(* CODESYS project oakslibrary.library
   Title: OaksLibrary
   Version: 1.1
   Placeholder: OaksLibrary
   Company: OaksAB

Project tree, tasks and I/O mapping:
  libraries: Tc2_BA, 3.3.9.0 (Beckhoff Automation GmbH); Tc2_EtherCAT, * (Beckhoff Automation GmbH); Tc2_IoFunctions, 3.3.13.0 (Beckhoff Automation GmbH); Tc2_Standard, 3.3.3.0 (Beckhoff Automation GmbH); Tc2_SUPS, 3.3.8.0 (Beckhoff Automation GmbH); Tc2_System, 3.4.24.0 (Beckhoff Automation GmbH); Tc2_SystemCX, 3.3.6.0 (Beckhoff Automation GmbH); Tc2_Utilities, * (Beckhoff Automation GmbH); Tc3_BA, 1.1.5.0 (Beckhoff Automation GmbH); Tc3_BA_Common, 2.1.4.0 (Beckhoff Automation GmbH); Tc3_Module, 3.3.21.0 (Beckhoff Automation GmbH)
  oaksLibrary/
    1 Ej vidareutveckling/
      function block fbDewpoint [ST]
      function block fbModbusSekvens [ST]
      function fRealToHour [CFC]
      function fRealToMinute [CFC]
      function fRealToSecond [CFC]
    Beräkning/
      Närvaro/
        function block fbCalcPresenceCo2Flow [ST]
        function fCalcPresenceCo2Flow [ST]
      function fAverageValueCalc [ST]
      function block fbCopCalc [ST]
      function block fbDewpointCalc [ST]
      function block fbDewPointSafe [ST]
      function block fbDifferenceCheck [ST]
      function block fbHeatExhEfficiency [ST]
      function block fbHourDiff [ST]
      function block fbMeanValueBC [ST]
      function block fbOperatingHours [ST]
      function block fbScale6pSupTempRad [ST]
      function block fbScale6pSuptempVent [ST]
      function block fbSfpCalc [ST]
      function block fbSunClock [ST]: DAY_OF_YEAR, DEG, FLOOR2, HOUR, HOUR_TO_TIME, HOUR_TO_TOD, MINUTE, MODR, mPercentageOfDay, mSolnedOchUppGangForskjuten, mSoluppgangOchSolnedgang, RAD, SUN_MIDDAY
      function fCalcFlow [ST]
      function fCalcFlowfbNicotraGerbhardtRLM [ST]
      function fScale12pInternalSetpoint [ST]
      function fScale20p [ST]
      function fScale2p [ST]
      function fScale2pInternalSetpoint [ST]
      function fScale3p [ST]
      function fScale3pInternalSetpoint [ST]
      function fScale6p [ST]
      function fScale6pInternalSetpoint [ST]
      function fScale7p [ST]
      function fScale7pInternalSetpoint [ST]
    Brand/
      function block fbFirealarm [ST]
      function block fbFirealarmFailure [ST]
      function block fbFireDamper [ST]
      function block fbFireDamperEvac [ST]
      function block fbFiredamperExercise [ST]
      function block fbFireDamperOneInput [ST]
      function block fbFireDamperWithAnalogOutput [ST]
      function block fbSmokeDetector [ST]
    Börvärden/
      function block fbPowerLimiter [ST]
      function block fbRoomCompensation [ST]
      function block fbSetPointBase [ST]
      function block fbSetPointC [ST]
      function block fbSetPointCMinMax [ST]
      function block fbSetPointKpa [ST]
      function block fbSetPointLs [ST]
      function block fbSetPointOutdoorCompC [ST]: mBv
      function block fbSetPointOutdoorCompkPa [ST]: mBv
      function block fbSetPointOutdoorCompLs [ST]: mBv
      function block fbSetPointOutdoorCompPa [ST]: mBv
      function block fbSetPointPa [ST]
      function block SetPointOutdoorCompCDewpoint [ST]
    Datahantering/
      function F_GetTempToUse [ST]
      function F_GetTempToUseMeanTemp [ST]
      function block FbDoubleControlledVariable [ST]
      function block FbDoubleControlledVariableLreal [ST]
      function block FbDoubleControlledVariableReal [ST]
      function block FbDoubleControlledVariableRealToWord [ST]
      function block FbDoubleControlledVariableWord [ST]
      function block fbModbusSekvensArray [ST]: mModbusSekvens, mModbusSekvensUppTill1000
      function fDwordToWordHigh [ST]
      function fDwordToWordLow [ST]
      function fRealToWord [ST]
      function fSetpointLimiter [ST]
      function fSignedConverter [ST]
      function fSignedDoubleConverter [ST]
      function fWordToDoubleWord [ST]
      data type uRealToTwoWORD
    DUTs/
      data type ST_ValueEnableError
    EtherCAT Specifikt/
      Givare/
        function block fbOutDoorTempMeanEL3204 [ST]: mMean
        function block fbPtEL3204 [ST]
      System/
        function block fbOaksSystemEtherCAT [ST]
    Familjebostäder/
      function block fbMotorRadFamiljebostader [ST]
    Givare/
      function block fbGeneralSensor [ST]
      function block fbOutDoorTempMean [ST]: mMean
      function block fbOutDoorTempMeanLuxLightCon [ST]: mMean, mPv
      function block fbPT1000 [ST]: mPv
      function block fbVoltage [ST]
      function block fbVoltageBar [ST]
      function block fbVoltageCo [ST]
      function block fbVoltageCo2 [ST]
      function block fbVoltagekPa [ST]
      function block fbVoltageLs [ST]
      function block fbVoltageLux [ST]
      function block fbVoltageLuxLightCon [ST]
      function block fbVoltageNo2 [ST]
      function block fbVoltagePa [ST]
      function block fbVoltagePaFlowLs [ST]
      function block fbVoltageRh [ST]
      function block fbVoltageTemp [ST]
      function block fbVoltageTempCo2 [ST]
      function block fbVoltageTempRh [ST]
    Hämta värde från Webport/
      function block fbOutDoorTempMeanFromScada [ST]: mMean
    Larm/
      Larm med inbyggd larmtagg/
        function block fbFreezeAlarm [ST]
        function block fbFreezeAlarmVoltage [ST]
        function block fbFusealarm [ST]
        function block fbJfb [ST]
        function block fbLeakDetector [ST]
        function block fbManometerLow [ST]
        function block fbManometerLowHigh [ST]
        function block fbOvervoltageProtection [ST]
        function block fbRotationGuard [ST]
      function block fbAlarm [ST]
      function block fbDamperAlarmOneInput [ST]
      function block fbDevAlarm [ST]
      function block fbDigitalAlarmIO [ST]
      function block fbFloorheatHighTemp [ST]
      function block fbFreezeAlarmNoSensor [ST]
      function block fbHighLimitAlarm [ST]
      function block fbLowLimitAlarm [ST]
    Mätare/
      function block fbEnergyCounterCondition [ST]
      function block fbPulseMeterE_P [ST]
      function block fbPulseMeterkWh [ST]
      function block fbPulseMeterM3 [ST]
      function block fbPulseMeterMWh [ST]
      function block fbPulseMeterV_Q [ST]
      function block fbPulseMeterV_Q_E_P [ST]
    Omvandling/
      function fUdintToTime [ST]
    Poseidon/
      function block fbMotorRadMeanTempPoseidon [ST]: mStartPump
      function block fbPowerLimiterPoseidon [ST]
      function block fbRoomCompPoseidon [ST]: mIAktuelltDriftlage
    Regulatorer/
      Utökade regulatorer/
        function block fbAdvSequenceController2Stages [ST]: mContainsCoolingSequence, mCoolSetpointCheck, mDevAlarmCheck
        function block fbAdvSequenceController3Stages [ST]: mContainsCoolingSequence, mCoolSetpointCheck, mDevAlarmCheck
        function block fbAdvSequenceController4Stages [ST]: mContainsCoolingSequence, mCoolSetpointCheck, mDevAlarmCheck
        function block fbAdvSequenceController5Stages [ST]: mContainsCoolingSequence, mCoolSetpointCheck, mDevAlarmCheck
        function block fbAdvSequenceController6Stages [ST]: mContainsCoolingSequence, mCoolSetpointCheck, mDevAlarmCheck
        function block fbAdvSequenceController7Stages [ST]: mContainsCoolingSequence, mCoolSetpointCheck, mDevAlarmCheck
      function block fbController [ST]: mDevAlarmCheck
      function block fbSequenceController2Stages [ST]: mContainsCoolingSequence, mCoolSetpointCheck, mDevAlarmCheck
      function block fbSequenceController3Stages [ST]: mContainsCoolingSequence, mCoolSetpointCheck, mDevAlarmCheck
      function block fbSequenceController4Stages [ST]: mContainsCoolingSequence, mCoolSetpointCheck, mDevAlarmCheck
      function block fbSequenceController5Stages [ST]: mContainsCoolingSequence, mCoolSetpointCheck, mDevAlarmCheck
      function block fbSequenceController6Stages [ST]: mContainsCoolingSequence, mCoolSetpointCheck, mDevAlarmCheck
      function block fbSequenceController7Stages [ST]: mContainsCoolingSequence, mCoolSetpointCheck, mDevAlarmCheck
    Skicka värden mellan plc/
      Inbyggda taggar/
        function block fbReadAdsBoolGeneralWp [ST]
        function block fbReadAdsRealGeneralWp [ST]
        function block fbReadAdsRealOutdoorMeantempWp [ST]
        function block fbReadAdsRealOutdoortempWp [ST]
        function block fbReadAdsTempSensorWp [ST]
      function block fbReadADSBool [ST]
      function block fbReadAdsInt [ST]
      function block fbReadADSReal [ST]
      function block fbReadAdsRealOutdoortemp [ST]
    System/
      function block fbBK9050 [ST]
      function block fbHardwareModelInfo [ST]
      function block fbOaksSystem [ST]
      function block fbSumAlarmWp [ST]
    Utsignal DO_AO/
      Motorer/
        function block fbGenericMotorHeatCool [ST]
        function block fbMotor [ST]: mStartDelayRemaining, mStopDelayRemaining, mTimeRemainingTof, mTimeRemainingTon
        function block fbMotorAo [ST]: mAnalogOutputActiveWhenCmdIsTrue
        function block fbMotorAoCool [ST]
        function block fbMotorAoRad [ST]
        function block fbMotorAoRl [ST]
        function block fbMotorCool [ST]
        function block fbMotorHeatBattery [ST]
        function block fbMotorHiLoSpeed [ST]
        function block fbMotorRad [ST]
        function block fbTwinMotorControl [ST]
        function block fbTwinMotorControlCool [ST]
        function block fbTwinMotorControlRad [ST]
      Värmeväxling/
        Enskilda funktioner/
          function block fbCoolRecycleHeatExhanger [ST]
          function block fbHeatExchangerStartup [ST]
        Korsvärmeväxlare/
          function block fbCrossFlowHeatExchanger [ST]
          function block fbCrossFlowHeatExhTemp [ST]
        function block fbHeatExhange [ST]
        function block fbHeatExhangeEff [ST]
      function block fbAnalogSignalLogic [ST]
      function block fbAnalogSignalLogicFb [ST]
      function block fbComfoVent [ST]
      function block fbDigitalSignalLogic [ST]: mStartDelayRemaining, mStopDelayRemaining, mTimeRemainingTof, mTimeRemainingTon
      function block fbDigitalSignalLogicFb [ST]: mStartDelayRemaining, mStopDelayRemaining, mTimeRemainingTof, mTimeRemainingTon
      function block fbGeneralSignalLogic [ST]
      function block fbLightSignalLogic [ST]: mBelysningsvillkor
      function block fbLightSignalLogicLux [ST]: mBelysningsvillkor
      function fKx2652State [ST]
    Växlingsblock/
      function block fbDailyToggle [ST]
      function block fbMonthlyToggle [ST]
      function block fbToggleStep [ST]
      function block fbWeeklyToggle [ST]
    function block fbCoolPumpSr [ST]
    function block fbEdge [ST]
    function block fbExcerciseInactiveMotor [ST]
    function block fbHeatPumpSr [ST]
    function block fbHystReal [ST]
    function block fbNightCooling [ST]
    function block fbNightheating [ST]
    function block fbPresenceDetector [ST]
    function block fbPumpMotion [ST]
    function block fbPushButton [ST]
    function block fbResetButton [ST]
    function block fbServiceSwitch [ST]
    function block fbServiceSwitch01A [ST]
    function block fbTimeChannelWp [ST]
    function block fbToggle [ST]
    function block fbVentilationUnit [ST]: mDrifttidslarm
    function block fbWatchdogSwitching [ST]
    global variables oaksGVL
*)

// oaksLibrary/Datahantering/uRealToTwoWORD
TYPE uRealToTwoWORD :
UNION
	rTest : REAL;
	wTest : ARRAY [0..1] OF  WORD;

END_UNION
END_TYPE

// oaksLibrary/DUTs/ST_ValueEnableError
TYPE ST_ValueEnableError :
STRUCT
	bEnable : BOOL := FALSE; //Aktivering
	rValue : REAL; //Värde
	bError : BOOL := FALSE; //Generellt fel
END_STRUCT
END_TYPE

// oaksLibrary/oaksGVL
{attribute 'qualified_only'}
VAR_GLOBAL
	iYear 	: INT; // År (Uppdateras från fbOaksSystem-block)
	iMonth 	: INT; // Månad(1-12) (Uppdateras från fbOaksSystem-block)
	iDay 	: INT; // Dag (1-31) (Uppdateras från fbOaksSystem-block)
	iDayOfWeek		: INT; // Veckodag (1-7) (Uppdateras från fbOaksSystem-block)
	iHour 	: INT; // Timme (0-23) (Uppdateras från fbOaksSystem-block)
	iMinute 	: INT; // Minut (0-59) (Uppdateras från fbOaksSystem-block) 
	iHourAndMinute : INT; // (iHour * 100) + iMinute (Uppdateras från fbOaksSystem-block) 
	iSecond 	: INT; // Sekund (0-59)	(Uppdateras från fbOaksSystem-block)

	fbPassiveAnalogInConfigTonReset : TON; // Återställer bPassiveAnalogInConfig till FALSE efter 30 sekunder. Körs från fbSystem-block.
	bPassiveAnalogInConfig : BOOL; // Sätt denna till true för att ladda givarkonfiguration på analoga in io. Återställs automatiskt efter 30 sekunder.
	

	bSummalarm AT %Q*  : BOOL; // Tänds om någon instans av fbAlarm larmar
	bSummalarmEjAutoReset AT %Q*  : BOOL; // Tänds om någon instans av fbAlarm med icke autoresetande/självkvitterande larm larmar
	fbSummalarmTOF :TOF; // Internvariabel används av summalarmsblock
	fbSummalarmEjAutoResetTOF :TOF; // Internvariabel används av summalarmsblock	
	
	bWatchdog  : BOOL; //Watchdog script i webport växlar
	bFireAlarm : BOOL := TRUE; // Global brandlarmsvariabel. Sätts av blocket fbFirealarm
	
	aBModbusBusyFlagga : ARRAY [1..15,0..255] OF BOOL;
	aBModbusSekvens : ARRAY [1..16] OF INT := [1, 1, 1, 1, 1, 1, 1, 1, 1, 1 ];
	
	aBModbusBusyFlaggaAdresser : ARRAY [1..2,0..3000] OF BOOL; //Används när man har många läsningar till samma enhet (exempelvis elvaco tempgivare)
	
	itemp : INT;
	
	bSekvensstart1  : BOOL; //Sekvensstart 1  sätts till TRUE från fbOaksSystem efter inställd tid
	bSekvensstart2  : BOOL; //Sekvensstart 2  sätts till TRUE från fbOaksSystem efter inställd tid
	bSekvensstart3  : BOOL; //Sekvensstart 3  sätts till TRUE från fbOaksSystem efter inställd tid
	bSekvensstart4  : BOOL; //Sekvensstart 4  sätts till TRUE från fbOaksSystem efter inställd tid
	bSekvensstart5  : BOOL; //Sekvensstart 5  sätts till TRUE från fbOaksSystem efter inställd tid
	bSekvensstart6  : BOOL; //Sekvensstart 6  sätts till TRUE från fbOaksSystem efter inställd tid
	bSekvensstart7  : BOOL; //Sekvensstart 7  sätts till TRUE från fbOaksSystem efter inställd tid
	bSekvensstart8  : BOOL; //Sekvensstart 8  sätts till TRUE från fbOaksSystem efter inställd tid
	bSekvensstart9  : BOOL; //Sekvensstart 9  sätts till TRUE från fbOaksSystem efter inställd tid
	bSekvensstart10 : BOOL; //Sekvensstart 10 sätts till TRUE från fbOaksSystem efter inställd tid
	bSekvensstart11 : BOOL; //Sekvensstart 11 sätts till TRUE från fbOaksSystem efter inställd tid
	bSekvensstart12 : BOOL; //Sekvensstart 12 sätts till TRUE från fbOaksSystem efter inställd tid
	bSekvensstart13 : BOOL; //Sekvensstart 13 sätts till TRUE från fbOaksSystem efter inställd tid
	bSekvensstart14 : BOOL; //Sekvensstart 14 sätts till TRUE från fbOaksSystem efter inställd tid
	bSekvensstart15 : BOOL; //Sekvensstart 15 sätts till TRUE från fbOaksSystem efter inställd tid
	bSekvensstart16 : BOOL; //Sekvensstart 15 sätts till TRUE från fbOaksSystem efter inställd tid
	
	
	

	bEnableSekvens1 : BOOL := TRUE; //blockering sekvens1 modbus
	bEnableSekvens2 : BOOL := TRUE; //blockering sekvens2 modbus
	bEnableSekvens3 : BOOL := TRUE; //blockering sekvens3 modbus
	bEnableSekvens4 : BOOL := TRUE; //blockering sekvens4 modbus
	bEnableSekvens5 : BOOL := TRUE; //blockering sekvens5 modbus
	bEnableSekvens6 : BOOL := TRUE; //blockering sekvens6 modbus
	bEnableSekvens7 : BOOL := TRUE; //blockering sekvens7 modbus
	bEnableSekvens8 : BOOL := TRUE; //blockering sekvens8 modbus
	bEnableSekvens9 : BOOL := TRUE; //blockering sekvens9 modbus
	bEnableSekvens10 : BOOL := TRUE; //blockering sekvens10 modbus
	bEnableSekvens11 : BOOL := TRUE; //blockering sekvens11 modbus
	bEnableSekvens12 : BOOL := TRUE; //blockering sekvens12 modbus
	bEnableSekvens13 : BOOL := TRUE; //blockering sekvens13 modbus
	bEnableSekvens14 : BOOL := TRUE; //blockering sekvens14 modbus
	bEnableSekvens15 : BOOL := TRUE; //blockering sekvens15 modbus
	bEnableSekvens16 : BOOL := TRUE; //blockering sekvens16 modbus					
	
// gammal modbussekvens funktion ny är i ovanstående array
	aBModbusSekvens1 : INT := 1;
	aBModbusBusyFlagga1 : ARRAY [0..255] OF BOOL;
	aBModbusSekvens2 : INT := 1;
	aBModbusBusyFlagga2 : ARRAY [0..255] OF BOOL;
	aBModbusSekvens3 : INT := 1;
	aBModbusBusyFlagga3 : ARRAY [0..255] OF BOOL;
	aBModbusSekvens4 : INT := 1;
	aBModbusBusyFlagga4 : ARRAY [0..255] OF BOOL;
	aBModbusSekvens5 : INT := 1;
	aBModbusBusyFlagga5 : ARRAY [0..255] OF BOOL;
	aBModbusSekvens6 : INT := 1;
	aBModbusBusyFlagga6 : ARRAY [0..255] OF BOOL;
	aBModbusSekvens7 : INT := 1;
	aBModbusBusyFlagga7 : ARRAY [0..255] OF BOOL;
	aBModbusSekvens8 : INT := 1;
	aBModbusBusyFlagga8 : ARRAY [0..255] OF BOOL;
	aBModbusSekvens9 : INT := 1;
	aBModbusBusyFlagga9 : ARRAY [0..255] OF BOOL;
	aBModbusSekvens10 : INT := 1;
	aBModbusBusyFlagga10 : ARRAY [0..255] OF BOOL;
	
	rOutdoorTemp : REAL; // global utetemp sätts i blocket fbOutDoorTempMean
	rOutdoorTempErrorValue0 : REAL; // global utetemp som ställs till 0 vid givarfel sätts i blocket fbOutDoorTempMean.
	rOutdoorTempErrorValue150 : REAL; // global utetemp som ställs till 150 vid givarfel sätts i blocket fbOutDoorTempMean.
	rOutdoorTempMean : REAL; // global medel utetemp sätts i blocket fbOutDoorTempMean
	bOutdoorTempSensorError : BOOL; // Givarfel utegivare sätts i blocket fbOutDoorTempMean
	
	bReset : BOOL; //Reset förreglande larm
	bPumpMotion : BOOL;  // Global variabel för pumpmotion
	
	//OaksTree
	bOptimizeWatchdog : BOOL := FALSE; //Watch-dog för optimeringsfunktioner (OaksTree) sätts till 1.
	bOptimizeActivate : BOOL := FALSE; //Global blockering av optimeringsfunktioner (OaksTree)
	
	//Felräknare för implicit-kontroller
	udiCheckBounds			: UDINT := 0;	//Felräknare field bounds (index)	
	udiCheckDivDInt			: UDINT := 0;	//Felräknare DBZ INT/UINT
	udiCheckDivLInt			: UDINT := 0;	//Felräknare DBZ LINT/ULINT
	udiCheckDivLReal		: UDINT := 0;	//Felräknare DBZ LREAL
	udiCheckDivReal			: UDINT := 0;	//Felräknare DBZ REAL
	udiCheckLRangeSigned	: UDINT := 0;	//Felräknare range LINT
	udiCheckLRangeUnsigned	: UDINT := 0;	//Felräknare range ULINT
	udiCheckPointer			: UDINT := 0;	//Felräknare pointer
	udiCheckRangeSigned		: UDINT := 0;	//Felräknare range INT
	udiCheckRangeUnsigned	: UDINT := 0;	//Felräknare range UINT
END_VAR

// oaksLibrary/1 Ej vidareutveckling/fbDewpoint
//OAKS AB
//2020-05-05
//Funktionsblock för beräkning av daggpunktstemperatur via temperatur/fukt.
{attribute 'obsolete' := 'Använd ersättningsblock.'}
FUNCTION_BLOCK fbDewpoint
VAR_INPUT
	rTemperature : REAL;
	rRelativeHumidity : REAL;
	rSetpoint : REAL :=14; //Börvärde
END_VAR

VAR_OUTPUT
	{attribute 'OPC.UA.DA' := '1'}
	PV AT %M* : REAL; //Uträknad daggpunkt~wp:[unit]°C[format]0.0[trendoptions]i:300
	rCSP : REAL; //Uträknat börvärde (börvärde eller daggpunkt + 2)
END_VAR

VAR
	FB_BA_HX01 : Tc2_BA.FB_BA_HX;
END_VAR

VAR_INPUT PERSISTENT
	{attribute 'OPC.UA.DA' := '1'}
	SP1 AT %M* : REAL := 12; //Min.begränsning framledningstemperatur~wp:[unit]°C[format]0.0[trendoptions]i:300
	{attribute 'OPC.UA.DA' := '1'}
	SP2 AT %M* : REAL := 25; //Max.begränsning framledningstemperatur~wp:[unit]°C[format]0.0[trendoptions]i:300
END_VAR

	FB_BA_HX01(
	rT:= rTemperature, 
	rHumRel:= rRelativeHumidity, 
	rAP:= 1013.25, 
	lrHumAbs=> , 
	lrDewPnt=> , 
	lrE=> , 
	lrDHA=> , 
	lrSpecV=> , 
	lrTWet=> );
	
	PV := LREAL_TO_REAL(FB_BA_HX01.lrDewPnt);
	
	//Uträknat börvärde daggpunkt
	rCSP := LIMIT(SP1, MAX(rSetpoint, (PV+2)), SP2);

END_FUNCTION_BLOCK

// oaksLibrary/1 Ej vidareutveckling/fbModbusSekvens
// Block för sekvenshantering av modbus. Använder sig av globala variabler oaksgvl.aBModbusBusyFlaggaX oaksgvl.aBModbusSekvensX
// Finns 10 "slingor"
{attribute 'obsolete' := 'Använd ersättningsblock.'}
FUNCTION_BLOCK fbModbusSekvens
VAR_INPUT
END_VAR
VAR_OUTPUT
END_VAR
VAR
	iTemp : INT; // används för temporär lagring	

	TON01sekvens1 : TON;
	TON02sekvens1 : TON;
	
	TON01sekvens2 : TON;
	TON02sekvens2 : TON;
	
	TON01sekvens3 : TON;
	TON02sekvens3 : TON;

	TON01sekvens4 : TON;
	TON02sekvens4 : TON;
	
	TON01sekvens5 : TON;
	TON02sekvens5 : TON;
	
	TON01sekvens6 : TON;
	TON02sekvens6 : TON;
	
	TON01sekvens7 : TON;
	TON02sekvens7 : TON;
	
	TON01sekvens8 : TON;
	TON02sekvens8 : TON;
	
	TON01sekvens9 : TON;
	TON02sekvens9 : TON;
	
	TON01sekvens10 : TON;
	TON02sekvens10 : TON;
END_VAR



IF NOT oaksgvl.aBModbusBusyFlagga1[oaksgvl.aBModbusSekvens1] OR TON02sekvens1.Q THEN
	TON01sekvens1(IN:=TRUE , PT:=T#1S , Q=> , ET=> );
	TON02sekvens1(IN:=FALSE , PT:=T#5S , Q=> , ET=> );	
	IF TON01sekvens1.Q THEN
		iTemp := oaksgvl.aBModbusSekvens1;
		oaksgvl.aBModbusSekvens1 := iTemp + 1;
		IF oaksgvl.aBModbusSekvens1 = 100  THEN
			oaksgvl.aBModbusSekvens1 := 1;
		END_IF
	END_IF
ELSE
	TON01sekvens1(IN:=FALSE , PT:=T#1S , Q=> , ET=> );	
	TON02sekvens1(IN:=TRUE , PT:=T#5S , Q=> , ET=> );	
END_IF

IF NOT oaksgvl.aBModbusBusyFlagga2[oaksgvl.aBModbusSekvens2] OR TON02Sekvens2.Q THEN
	TON01Sekvens2(IN:=TRUE , PT:=T#1S , Q=> , ET=> );
	TON02Sekvens2(IN:=FALSE , PT:=T#5S , Q=> , ET=> );	
	IF TON01Sekvens2.Q THEN
		iTemp := oaksgvl.aBModbusSekvens2;
		oaksgvl.aBModbusSekvens2 := iTemp + 1;
		IF oaksgvl.aBModbusSekvens2 = 100  THEN
			oaksgvl.aBModbusSekvens2 := 1;
		END_IF
	END_IF
ELSE
	TON01Sekvens2(IN:=FALSE , PT:=T#1S , Q=> , ET=> );	
	TON02Sekvens2(IN:=TRUE , PT:=T#5S , Q=> , ET=> );	
END_IF

IF NOT oaksgvl.aBModbusBusyFlagga3[oaksgvl.aBModbusSekvens3] OR TON02Sekvens3.Q THEN
	TON01Sekvens3(IN:=TRUE , PT:=T#1S , Q=> , ET=> );
	TON02Sekvens3(IN:=FALSE , PT:=T#5S , Q=> , ET=> );	
	IF TON01Sekvens3.Q THEN
		iTemp := oaksgvl.aBModbusSekvens3;
		oaksgvl.aBModbusSekvens3 := iTemp + 1;
		IF oaksgvl.aBModbusSekvens3 = 100  THEN
			oaksgvl.aBModbusSekvens3 := 1;
		END_IF
	END_IF
ELSE
	TON01Sekvens3(IN:=FALSE , PT:=T#1S , Q=> , ET=> );	
	TON02Sekvens3(IN:=TRUE , PT:=T#5S , Q=> , ET=> );	
END_IF

IF NOT oaksgvl.aBModbusBusyFlagga4[oaksgvl.aBModbusSekvens4] OR TON02Sekvens4.Q THEN
	TON01Sekvens4(IN:=TRUE , PT:=T#1S , Q=> , ET=> );
	TON02Sekvens4(IN:=FALSE , PT:=T#5S , Q=> , ET=> );	
	IF TON01Sekvens4.Q THEN
		iTemp := oaksgvl.aBModbusSekvens4;
		oaksgvl.aBModbusSekvens4 := iTemp + 1;
		IF oaksgvl.aBModbusSekvens4 = 100  THEN
			oaksgvl.aBModbusSekvens4 := 1;
		END_IF
	END_IF
ELSE
	TON01Sekvens4(IN:=FALSE , PT:=T#1S , Q=> , ET=> );	
	TON02Sekvens4(IN:=TRUE , PT:=T#5S , Q=> , ET=> );	
END_IF

IF NOT oaksgvl.aBModbusBusyFlagga5[oaksgvl.aBModbusSekvens5] OR TON02Sekvens5.Q THEN
	TON01Sekvens5(IN:=TRUE , PT:=T#1S , Q=> , ET=> );
	TON02Sekvens5(IN:=FALSE , PT:=T#5S , Q=> , ET=> );	
	IF TON01Sekvens5.Q THEN
		iTemp := oaksgvl.aBModbusSekvens5;
		oaksgvl.aBModbusSekvens5 := iTemp + 1;
		IF oaksgvl.aBModbusSekvens5 = 100  THEN
			oaksgvl.aBModbusSekvens5 := 1;
		END_IF
	END_IF
ELSE
	TON01Sekvens5(IN:=FALSE , PT:=T#1S , Q=> , ET=> );	
	TON02Sekvens5(IN:=TRUE , PT:=T#5S , Q=> , ET=> );	
END_IF

IF NOT oaksgvl.aBModbusBusyFlagga6[oaksgvl.aBModbusSekvens6] OR TON02Sekvens6.Q THEN
	TON01Sekvens6(IN:=TRUE , PT:=T#1S , Q=> , ET=> );
	TON02Sekvens6(IN:=FALSE , PT:=T#5S , Q=> , ET=> );	
	IF TON01Sekvens6.Q THEN
		iTemp := oaksgvl.aBModbusSekvens6;
		oaksgvl.aBModbusSekvens6 := iTemp + 1;
		IF oaksgvl.aBModbusSekvens6 = 100  THEN
			oaksgvl.aBModbusSekvens6 := 1;
		END_IF
	END_IF
ELSE
	TON01Sekvens6(IN:=FALSE , PT:=T#1S , Q=> , ET=> );	
	TON02Sekvens6(IN:=TRUE , PT:=T#5S , Q=> , ET=> );	
END_IF

IF NOT oaksgvl.aBModbusBusyFlagga7[oaksgvl.aBModbusSekvens7] OR TON02Sekvens7.Q THEN
	TON01Sekvens7(IN:=TRUE , PT:=T#1S , Q=> , ET=> );
	TON02Sekvens7(IN:=FALSE , PT:=T#5S , Q=> , ET=> );	
	IF TON01Sekvens7.Q THEN
		iTemp := oaksgvl.aBModbusSekvens7;
		oaksgvl.aBModbusSekvens7 := iTemp + 1;
		IF oaksgvl.aBModbusSekvens7 = 100  THEN
			oaksgvl.aBModbusSekvens7 := 1;
		END_IF
	END_IF
ELSE
	TON01Sekvens7(IN:=FALSE , PT:=T#1S , Q=> , ET=> );	
	TON02Sekvens7(IN:=TRUE , PT:=T#5S , Q=> , ET=> );	
END_IF

IF NOT oaksgvl.aBModbusBusyFlagga8[oaksgvl.aBModbusSekvens8] OR TON02Sekvens8.Q THEN
	TON01Sekvens8(IN:=TRUE , PT:=T#1S , Q=> , ET=> );
	TON02Sekvens8(IN:=FALSE , PT:=T#5S , Q=> , ET=> );	
	IF TON01Sekvens8.Q THEN
		iTemp := oaksgvl.aBModbusSekvens8;
		oaksgvl.aBModbusSekvens8 := iTemp + 1;
		IF oaksgvl.aBModbusSekvens8 = 100  THEN
			oaksgvl.aBModbusSekvens8 := 1;
		END_IF
	END_IF
ELSE
	TON01Sekvens8(IN:=FALSE , PT:=T#1S , Q=> , ET=> );	
	TON02Sekvens8(IN:=TRUE , PT:=T#5S , Q=> , ET=> );	
END_IF

IF NOT oaksgvl.aBModbusBusyFlagga9[oaksgvl.aBModbusSekvens9] OR TON02Sekvens9.Q THEN
	TON01Sekvens9(IN:=TRUE , PT:=T#1S , Q=> , ET=> );
	TON02Sekvens9(IN:=FALSE , PT:=T#5S , Q=> , ET=> );	
	IF TON01Sekvens9.Q THEN
		iTemp := oaksgvl.aBModbusSekvens9;
		oaksgvl.aBModbusSekvens9 := iTemp + 1;
		IF oaksgvl.aBModbusSekvens9 = 100  THEN
			oaksgvl.aBModbusSekvens9 := 1;
		END_IF
	END_IF
ELSE
	TON01Sekvens9(IN:=FALSE , PT:=T#1S , Q=> , ET=> );	
	TON02Sekvens9(IN:=TRUE , PT:=T#5S , Q=> , ET=> );	
END_IF

IF NOT oaksgvl.aBModbusBusyFlagga10[oaksgvl.aBModbusSekvens10] OR TON02Sekvens10.Q THEN
	TON01Sekvens10(IN:=TRUE , PT:=T#1S , Q=> , ET=> );
	TON02Sekvens10(IN:=FALSE , PT:=T#5S , Q=> , ET=> );	
	IF TON01Sekvens10.Q THEN
		iTemp := oaksgvl.aBModbusSekvens10;
		oaksgvl.aBModbusSekvens10 := iTemp + 1;
		IF oaksgvl.aBModbusSekvens10 = 100  THEN
			oaksgvl.aBModbusSekvens10 := 1;
		END_IF
	END_IF
ELSE
	TON01Sekvens10(IN:=FALSE , PT:=T#1S , Q=> , ET=> );	
	TON02Sekvens10(IN:=TRUE , PT:=T#5S , Q=> , ET=> );	
END_IF

END_FUNCTION_BLOCK

// oaksLibrary/1 Ej vidareutveckling/fRealToHour
// Funktion för att omvandla inställingsvärde minuter från webport till TIME
{deprecated := 'Använd fUDintToTime istället'}
FUNCTION fRealToHour : TIME
VAR_INPUT
	rHour : REAL;
END_VAR
VAR

END_VAR

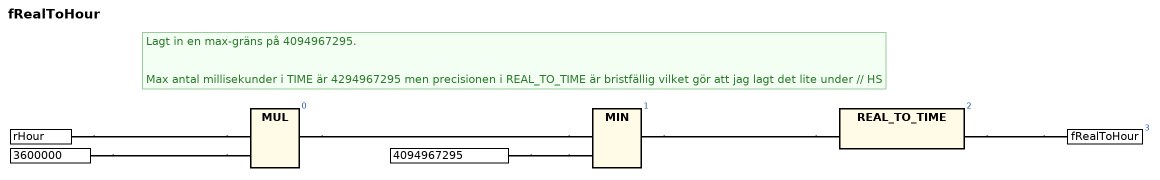
// Lagt in en max-gräns på 4094967295.
//
// Max antal millisekunder i TIME är 4294967295 men precisionen i REAL_TO_TIME är bristfällig vilket gör att jag lagt det lite under // HS
fRealToHour := REAL_TO_TIME(MIN(rHour * 3600000, 4094967295));

END_FUNCTION

// oaksLibrary/Omvandling/fUdintToTime
//Omvandlar en UDINT till TIME enligt vald tidsenhet
//Henrik H, 25-03-31
//Justerad Robert H, 25-03-31
FUNCTION fUdintToTime : TIME
VAR_INPUT
	byUnit : BYTE := 1;    	// Val av enhet (0 = ms, 1 = sekunder, 2 = minuter, 3 = timmar) (default sekunder)
    udiInputTime : UDINT; 	// UDINT som skall konverteras till vald TIME-enhet
END_VAR

VAR
    tResult : TIME;
END_VAR

CASE byUnit OF
	0: tResult := UDINT_TO_TIME(udiInputTime);                   	// Millisekunder
	1: tResult := UDINT_TO_TIME(udiInputTime * 1000);       		// Sekunder 
	2: tResult := UDINT_TO_TIME(udiInputTime * 60000);       		// Minuter
	3: tResult := UDINT_TO_TIME(udiInputTime * 3600000);			// Timmar
ELSE tResult := T#0S; 				                      			// Om ogiltigt val
END_CASE;
    
fUdintToTime := tResult;

END_FUNCTION

// oaksLibrary/1 Ej vidareutveckling/fRealToMinute
// Funktion för att omvandla inställingsvärde minuter från webport till TIME
{deprecated := 'Använd fUDintToTime istället'}
FUNCTION fRealToMinute : TIME
VAR_INPUT
	rMinute : REAL;
END_VAR
VAR
	lrTempReal : LREAL;
END_VAR

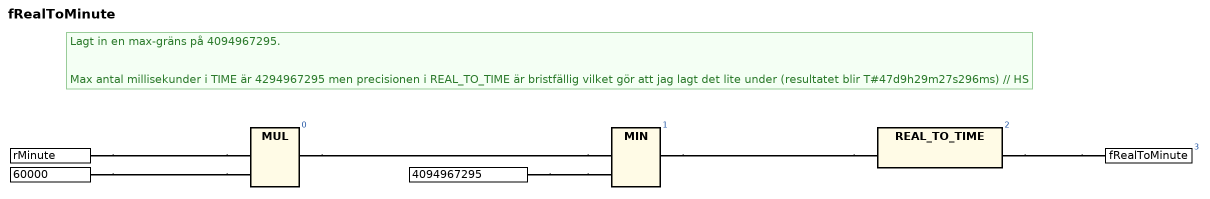
// Lagt in en max-gräns på 4094967295.
//
// Max antal millisekunder i TIME är 4294967295 men precisionen i REAL_TO_TIME är bristfällig vilket gör att jag lagt det lite under (resultatet blir T#47d9h29m27s296ms) // HS
fRealToMinute := REAL_TO_TIME(MIN(rMinute * 60000, 4094967295));

END_FUNCTION

// oaksLibrary/1 Ej vidareutveckling/fRealToSecond
// Funktion för att omvandla inställingsvärde sekunder från webport till TIME
{deprecated := 'Använd fUDintToTime istället'}
FUNCTION fRealToSecond : TIME
VAR_INPUT
	rSecond : REAL;
END_VAR
VAR
END_VAR

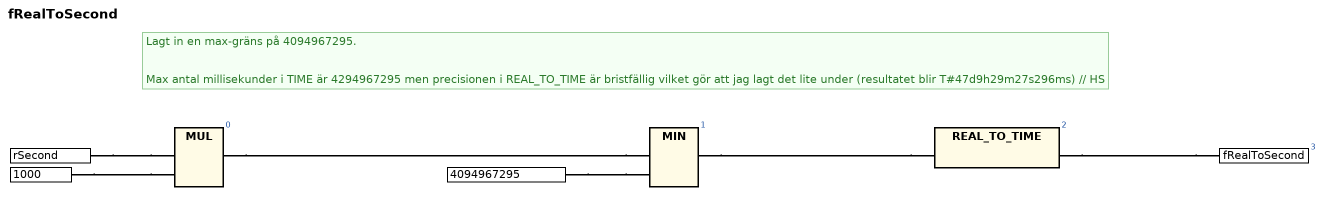
// Lagt in en max-gräns på 4094967295.
//
// Max antal millisekunder i TIME är 4294967295 men precisionen i REAL_TO_TIME är bristfällig vilket gör att jag lagt det lite under (resultatet blir T#47d9h29m27s296ms) // HS
fRealToSecond := REAL_TO_TIME(MIN(rSecond * 1000, 4094967295));

END_FUNCTION

// oaksLibrary/Beräkning/Närvaro/fbCalcPresenceCo2Flow
//Oaks AB
//2022-06-014
//Funktionsblock för att beräkna närvaro via co2/flöde med inbyggda taggar för visning i Webport.
//Till-/frånslagsfördröjning är inställbar.
FUNCTION_BLOCK fbCalcPresenceCo2Flow
VAR_INPUT
	rFlowLs : REAL; //Flöde i l/s
	rCo2 : REAL; //Koldioxidhalt	
END_VAR
VAR_INPUT PERSISTENT
	SP1 AT %M*: REAL := 0; //Gräns antal personer för närvaro 0=Avaktiverad~wp:[unit]st[format]0
	SP2 AT %M*: REAL := 0; //Tillslagsfördröjning närvaro~wp:[unit]min[format]0
	SP3 AT %M*: REAL := 0; //Frånslagsfördröjning närvaro~wp:[unit]min[format]0
END_VAR
VAR_OUTPUT
	PV AT %M*: REAL; //Antal personer~wp:[unit]st[format]0
	V AT %M*: BOOL; //Närvaro~wp:[trendoptions]i:14400, t:1
END_VAR
VAR
	bPresenceInternal : BOOL;
	TON_startDel: TON;
	TOF_StopDel: TOF;
END_VAR

//Calculate number of people in room
PV := fCalcPresenceCo2Flow(rFlowLs, rCo2);

//Check if detection is active
IF SP1 > 0 AND PV >= SP1 THEN
	bPresenceInternal := TRUE;
ELSE
	bPresenceInternal := FALSE;
END_IF

//Start Delay
TON_startDel(IN:= bPresenceInternal, PT:= fRealToMinute(SP2), Q=> , ET=> );

//Stop delay
TOF_StopDel(IN:= TON_startDel.Q, PT:= fRealToMinute(SP3), Q=> , ET=> );

//Indication
V := TON_startDel.Q OR (TOF_StopDel.Q AND NOT TON_startDel.Q);

END_FUNCTION_BLOCK

// oaksLibrary/Beräkning/Närvaro/fCalcPresenceCo2Flow
//Oaks AB
//2022-06-014
//Funktion för att beräkna närvaro via co2/flöde.
FUNCTION fCalcPresenceCo2Flow : REAL;
VAR_INPUT
	rFlowLs : REAL; //Flöde i l/s
	rCo2 : REAL; //Koldioxidhalt	
END_VAR
VAR
	rFlowInternal : REAL;
END_VAR

//Calculate number of people
rFlowInternal := ((3.6*rFlowLs)*(rCo2-410))/(24*1000); 
//Prevent negative values
fCalcPresenceCo2Flow := MAX(0,rFlowInternal);

END_FUNCTION

// oaksLibrary/Beräkning/fAverageValueCalc
//Oaks AB
//2022-07-14
//Funktion för medelvärdesberäkning och visning av min-/max värden för upp till 100 värden.
//Värden som inte är aktiverade (bEnable) har fel (bError) eller som är utanför gränsvärden (rLowLimit/rHighLimit) räknas bort ut medelvärdesberäkning.
//bErrorNoValues indikerar att inga giltliga värden finns
//ST_ValueEnableError kopplas till aValueArray (struct)

FUNCTION fAverageValueCalc : REAL
VAR_INPUT
	aValueArray: ARRAY[1..100] OF ST_ValueEnableError;
	rLowLimit : REAL := -50; //Låg gräns mätvärde
	rHighLimit : REAL := 10000; //Hög gräns mätvärde
END_VAR
VAR_OUTPUT
	//rAverageValue : LREAL; //Medelvärde
	rMinValue : REAL; //Lägsta värde
	rMaxValue : REAL; //Högsta värde
	iValidValues : UINT; //Giltliga värden
	iInvalidValues : UINT; //Ogiltliga värden
	bErrorNoValues : BOOL; //Inga giltliga värden
	bErrorInvalidValues : BOOL; //Ogiltliga värden förekommer
END_VAR
VAR
	nCounter : INT;
	rSum : LREAL;
	rMinInternal : REAL;
	rMaxInternal : REAL;
	bInitMinMax: BOOL;
	iSensorsWithError : UINT;
END_VAR

iValidValues := 0;
rSum := 0;
bInitMinMax := FALSE;
rMinInternal := 0;
rMaxInternal := 0;
iSensorsWithError := 0;

//Average
FOR nCounter := 1 TO 100 BY 1 DO

    //Not enabled
	IF NOT aValueArray[nCounter].bEnable THEN
		iValidValues := iValidValues;
		rSum := rSum;
	//Enabled but error occurs or values is out of boundaries
	ELSIF aValueArray[nCounter].bEnable AND (aValueArray[nCounter].bError OR aValueArray[nCounter].rValue <= rLowLimit OR aValueArray[nCounter].rValue >= rHighLimit) THEN
		iValidValues := iValidValues;
		rSum := rSum;
		iSensorsWithError := iSensorsWithError +1;
	//Value is valid
	ELSE
		iValidValues := iValidValues + 1;
		rSum := rSum + aValueArray[nCounter].rValue;
		
		//Init min/max (Only done once per cycle)
		IF NOT bInitMinMax THEN
			bInitMinMax := TRUE;
			rMinInternal := aValueArray[nCounter].rValue;
			rMaxInternal := aValueArray[nCounter].rValue;
		ELSE
			//Set min/max
			IF aValueArray[nCounter].rValue <= rMinInternal THEN 
				rMinInternal := aValueArray[nCounter].rValue;
			ELSE 
				rMinInternal := rMinInternal;
			END_IF
		
			IF aValueArray[nCounter].rValue >= rMaxInternal THEN 
				rMaxInternal := aValueArray[nCounter].rValue;
			ELSE 
				rMaxInternal := rMaxInternal;
			END_IF

		END_IF
		
	END_IF

END_FOR;

//Calculate Average if validsensors is larger than 0 else set error
IF iValidValues > 0 THEN
	fAverageValueCalc := rSum / iValidValues;
	bErrorNoValues := FALSE;
ELSE 
	fAverageValueCalc := 0;
	bErrorNoValues := TRUE;
END_IF

//Set min-/max values
rMinValue := rMinInternal;
rMaxValue := rMaxInternal;

//Invalid values
iInvalidValues := iSensorsWithError;
IF iInvalidValues > 0 THEN
	bErrorInvalidValues := TRUE;
ELSE
	bErrorInvalidValues := FALSE;
END_IF

END_FUNCTION

// oaksLibrary/Beräkning/fbCopCalc
// COP-kalkylering. Räknar ut förbrukning och produktion de senaste 24 timmarna och beräknar utifrån det COP-värde
FUNCTION_BLOCK fbCopCalc
VAR_INPUT
	rTotalConsumedEnergy : REAL; //Totalt förbrukad energi
	rTotalProducedEnergy : REAL; //Totalt producerad energi
END_VAR
VAR_OUTPUT
	rEnergyConsumedEnergyDiff: REAL; //Förbrukad energi senaste dygn
	rEnergyProducedEnergyDiff: REAL; //Producerad energi senaste dygn
	rCop 		: REAL; // aktuell cop
END_VAR
VAR
	FB_BA_GetTime01 : tc2_ba.FB_BA_GetTime; 
	FB_BA_ExtTiSt01 : tc2_ba.FB_BA_ExtTiSt;
	wMinute : WORD;
	fbMinuteTrig : R_TRIG;
	iTemp : INT;
	iCounter : INT;
END_VAR
VAR PERSISTENT
	wLastMinuteOfChange  : WORD;
	rArrayConsumedEnergy : ARRAY [0..1439] OF REAL;
	rArrayProducedEnergy : ARRAY [0..1439] OF REAL;
END_VAR

	FB_BA_GetTime01(bEn :=TRUE);	
	FB_BA_ExtTiSt01(stTi := FB_BA_GetTime01.stSysTi );

	IF FB_BA_ExtTiSt01.wMinute <> wLastMinuteOfChange THEN
		fbMinuteTrig(CLK := TRUE);
	ELSE
		fbMinuteTrig(CLK := FALSE);
	END_IF
	
	IF fbMinuteTrig.Q THEN
		FOR iCounter:=1439 TO 1 BY -1 DO
			rArrayConsumedEnergy[iCounter]:=rArrayConsumedEnergy[iCounter-1];
			rArrayProducedEnergy[iCounter]:=rArrayProducedEnergy[iCounter-1];
		END_FOR;
		rArrayConsumedEnergy[0] := rTotalConsumedEnergy;
		rArrayProducedEnergy[0] := rTotalProducedEnergy;
		wLastMinuteOfChange := FB_BA_ExtTiSt01.wMinute;
	END_IF 

	rEnergyConsumedEnergyDiff := rArrayConsumedEnergy[0] - rArrayConsumedEnergy[59]; 
	rEnergyProducedEnergyDiff := rArrayProducedEnergy[0] - rArrayProducedEnergy[59];

	IF rArrayConsumedEnergy[0] <> 0 AND rArrayProducedEnergy[0] <> 0 THEN
		rCop :=  rEnergyProducedEnergyDiff / rEnergyConsumedEnergyDiff;
	END_IF

END_FUNCTION_BLOCK

// oaksLibrary/Beräkning/fbDewpointCalc
//OAKS AB
//2020-05-05
//Funktionsblock för beräkning av daggpunktstemperatur via temperatur/fukt.
FUNCTION_BLOCK fbDewpointCalc
VAR_INPUT
	rTemperature : REAL;
	rRelativeHumidity : REAL;
	rSetpoint : REAL :=14; //Börvärde
	rSetpointOffest : REAL; //Börvärdesförskjutning över uträknad daggpunkt
END_VAR

VAR_OUTPUT
	{attribute 'OPC.UA.DA' := '1'}
	PV AT %M* : REAL; //Uträknad daggpunkt~wp:[unit]°C[format]0.0[trendoptions]i:300
	rCSP : REAL; //Uträknat börvärde (börvärde eller daggpunkt + 2)
END_VAR

VAR
	FB_BA_HX01 : Tc2_BA.FB_BA_HX;
END_VAR

	FB_BA_HX01(
	rT:= rTemperature, 
	rHumRel:= rRelativeHumidity, 
	rAP:= 1013.25, 
	lrHumAbs=> , 
	lrDewPnt=> , 
	lrE=> , 
	lrDHA=> , 
	lrSpecV=> , 
	lrTWet=> );
	
	PV := LREAL_TO_REAL(FB_BA_HX01.lrDewPnt);
	
	//Uträknat börvärde daggpunkt
	rCSP := MAX(rSetpoint, (PV+rSetpointOffest));

END_FUNCTION_BLOCK

// oaksLibrary/Beräkning/fbDewPointSafe
//OAKS AB
//2023-10-31
//Funktionsblock för beräkning av daggpunktstemperatur via temperatur/fukt.
//bSafe väljer ett fast säkert börvärde. Villkor ska te x vara givarfel/orimligt värde på temp/fukt
FUNCTION_BLOCK fbDewpointSafe
VAR_INPUT
	rTemperature : REAL;
	rRelativeHumidity : REAL;
	rSetpoint : REAL :=14; //Börvärde
	bSafe : BOOL; //Väljer SP3 som fast börvärde vid true
END_VAR

VAR_OUTPUT
	{attribute 'OPC.UA.DA' := '1'}
	PV AT %M* : REAL; //Uträknad daggpunkt~wp:[unit]°C[format]0.0[trendoptions]i:300
	rCSP : REAL; //Uträknat börvärde (börvärde eller daggpunkt + 2)
	AL AT %M* : BOOL; //Beräkningsfel, säkert börvärde används~wp:
END_VAR

VAR
	FB_BA_HX01 : Tc2_BA.FB_BA_HX;
	fbAlarm1 : fbAlarm;
END_VAR

VAR_INPUT PERSISTENT
	{attribute 'OPC.UA.DA' := '1'}
	SP1 AT %M* : REAL := 12; //Min.begränsning framledningstemperatur~wp:[unit]°C[format]0.0[trendoptions]i:300
	{attribute 'OPC.UA.DA' := '1'}
	SP2 AT %M* : REAL := 25; //Max.begränsning framledningstemperatur~wp:[unit]°C[format]0.0[trendoptions]i:300
	{attribute 'OPC.UA.DA' := '1'}
	SP3 AT %M* : REAL := 25; //Säkert börvärde vid ber.fel~wp:[unit]°C[format]0.0[trendoptions]i:300
END_VAR

	FB_BA_HX01(
	rT:= rTemperature, 
	rHumRel:= rRelativeHumidity, 
	rAP:= 1013.25, 
	lrHumAbs=> , 
	lrDewPnt=> , 
	lrE=> , 
	lrDHA=> , 
	lrSpecV=> , 
	lrTWet=> );
	
	PV := LREAL_TO_REAL(FB_BA_HX01.lrDewPnt);
	
	//Uträknat börvärde daggpunkt (välj SP3 vid bSafe)
	rCSP := SEL(bSafe, LIMIT(SP1, MAX(rSetpoint, (PV+2)), SP2), SP3);
	
	//Larm beräkningsfel
	fbAlarm1(bInput := bSafe, bAutoReset := TRUE, bAlarmOutput => AL);

END_FUNCTION_BLOCK

// oaksLibrary/Larm/fbAlarm
// Grundblock för larm används alltid vid programmering av larm då det triggar summalarmslampa
FUNCTION_BLOCK fbAlarm
VAR_INPUT
	bInput : BOOL; // larmvillkor
	tAlarmDelay : TIME := T#5S; // larmfördröjning
	bAutoReset : BOOL := TRUE; //autokvittering av larm
END_VAR
VAR_OUTPUT
	bAlarmOutput : BOOL; //larmutgång
END_VAR
VAR
	
	bAlarmFlag : BOOL;
	iTemp : INT;
	fbAlarmTon : TON;
	
	
	fbRestartFlagToN : TON;
	bRestartFlag : BOOL := TRUE;
	
END_VAR

fbAlarmTon.PT := tAlarmDelay;

fbRestartFlagToN.PT := T#5S;
fbRestartFlagToN(IN:=TRUE);
IF fbRestartFlagToN.Q THEN 
	bRestartFlag := FALSE;
END_IF



IF 	bInput AND NOT bRestartFlag THEN
	bAlarmFlag := TRUE;
ELSIF (NOT bInput AND bAutoReset) OR (NOT bInput AND (oaksGVL.bReset OR NOT bAlarmOutput)) THEN
	bAlarmFlag := FALSE;
END_IF

IF bAlarmFlag THEN
	fbAlarmTon(IN:= TRUE);
ELSE
	fbAlarmTon(IN:=FALSE );	
END_IF

bAlarmOutput := fbAlarmTon.Q;

// Tillägg för summalarmslampa
oaksGVL.fbSummalarmTOF.PT := T#5S;
oaksGVL.fbSummalarmTOF.IN := bAlarmOutput;
oaksGVL.fbSummalarmTOF();
oaksGVL.bSummalarm := oaksGVL.fbSummalarmTOF.Q;

// Tillägg för summalarmslampa för ej självkvitterande larm
oaksGVL.fbSummalarmEjAutoResetTOF.PT := T#1S;
oaksGVL.fbSummalarmEjAutoResetTOF.IN := bAlarmOutput AND NOT bAutoReset;
oaksGVL.fbSummalarmEjAutoResetTOF();
oaksGVL.bSummalarmEjAutoReset := oaksGVL.fbSummalarmEjAutoResetTOF.Q;

END_FUNCTION_BLOCK

// oaksLibrary/Beräkning/fbDifferenceCheck
// Funktionsblock som används för att kolla om senaste inlästa värde skiljer sig från föregående inläst.
FUNCTION_BLOCK fbDifferenceCheck
VAR_INPUT
	rPv : REAL;
END_VAR
VAR_OUTPUT
	bDifference : BOOL; // Blir till om insignal skiljer sig från förra cykel
END_VAR
VAR
	rInternalPv : REAL;
END_VAR

IF rPv <> rInternalPv THEN
	rInternalPv := rPv;
	bDifference := TRUE;
ELSE
	bDifference := FALSE;
END_IF

END_FUNCTION_BLOCK

// oaksLibrary/Beräkning/fbHeatExhEfficiency
//Funktionsblock för att beräkna verkningsgrad i ventilationsaggregat. Larm låg/hög verkninsgrad
//Verkningsgrad = (Tilluft efter VVX - Uteluft) / (Frånluft - Uteluft)
//Verkningsgrad = (Frånluft efter VVX - Avluft) / (Frånluft - Uteluft)
FUNCTION_BLOCK fbHeatExhEfficiency
VAR_INPUT
bSupfanInd : BOOL; // Driftindikering tilluftsfläkt
bCoolRecycle : BOOL ; // Aktiv kylåtervinning
rProcessValue : REAL; // Insignal från regulator
rSupTemp : REAL; // Tilluftstemperatur efter VVX
rOutdoorTemp : REFERENCE TO REAL; //Uteluftstemperatur Knyter man inget här används oaksGVL.rOutdoortemp
rExhTemp : REAL; // Frånluftstemperatur
rExhaustTemp : REAL; // Avluftstemperatur
bType : BOOL; // TRUE = Tilluft efter VVX/frånluft/uteluft FALSE= Frånluft/avluft/uteluft
END_VAR
VAR_OUTPUT
	{attribute 'OPC.UA.DA' := '1'}
	PV AT %M* : REAL; //Verkningsgrad~wp:[unit]%[format]0[trendoption]i:300
	{attribute 'OPC.UA.DA' := '1'}
	LAL AT %M* : BOOL; //Låg verkningsgrad~wp:
	{attribute 'OPC.UA.DA' := '1'}
	HAL AT %M* : BOOL; //Hög verkningsgrad~wp:
END_VAR
VAR
	rTempUsed : REAL; // Uteluftstemperatur
	//rTempUsed : REAL;
	rEff : REAL;	
	rTemp : REAL; // Tempvariablel
	fbLowEffeciency : fbLowLimitAlarm;
	fbHighEffeciency : fbHighLimitAlarm;
	bCalcAtive : BOOL;
END_VAR
VAR_INPUT PERSISTENT
{attribute 'OPC.UA.DA' := '1'}
AD AT %M* : INT :=60;//Larmfördröjning~wp:[unit]minuter[format]0
{attribute 'OPC.UA.DA' := '1'}
ALL AT %M* : INT :=30;  //Låg gräns verkningsgrad~wp:[unit]%[format]0
{attribute 'OPC.UA.DA' := '1'}
AHL AT %M* : INT :=90;  //Hög gräns verkningsgrad~wp:[unit]%[format]0
{attribute 'OPC.UA.DA' := '1'}
SP1 AT %M* : REAL :=0;//Beräkna verkningsgrad då utsignal överstiger~wp:[unit]%[format]0
END_VAR

//Temp select
	IF __ISVALIDREF(rOutdoorTemp) THEN
		rTempUsed := rOutdoorTemp;
	ELSE
		rTempUsed := oaksGVL.rOutdoorTemp;
	END_IF
		
// Verkningsgradsberäkning
rTemp := rExhTemp-rTempUsed;

//Hantering min/max begräsning för beräkning
IF SP1 < 0 THEN
	SP1 := 0;
ELSIF SP1 > 100 THEN
	SP1 := 100;
END_IF

//Aktivering av beräkning
IF rProcessValue >= SP1 THEN
	bCalcAtive := TRUE;
ELSE
	bCalcAtive := FALSE;
END_IF;

IF bType AND rTemp <> 0 AND NOT bCoolRecycle AND bSupfanInd AND bCalcAtive THEN
	rEff := ((rSupTemp-rTempUsed)/rTemp)*100;
ELSIF bType = FALSE AND rTemp <> 0 AND NOT bCoolRecycle AND bSupfanInd AND bCalcAtive THEN
	rEff := ((rExhTemp-rExhaustTemp)/rTemp)*100;
ELSIF bCoolRecycle OR NOT bSupfanInd OR NOT bCalcAtive THEN
	rEff := 0;
END_IF

IF rEff > 100 THEN
	PV := 100;
ELSIF rEff < 0 THEN
	PV := 0;
ELSE
	PV := rEff;
END_IF

// Larmfunktion låg/hög verkningsgrad
fbLowEffeciency(
	//bInput:= , 
	tAlarmDelay:= INT_TO_TIME(AD)*60000, 
	bAutoReset:=TRUE, 
	bAlarmOutput=>LAL, 
	bEnable:= rProcessValue > 100, 
	rProcessValue:=PV, 
	rLowLimit:=ALL
);
fbHighEffeciency(
	//bInput:= , 
	tAlarmDelay:= INT_TO_TIME(AD)*60000, 
	bAutoReset:= TRUE, 
	bAlarmOutput=>HAL , 
	bEnable:= rProcessValue > 100, 
	rProcessValue:=PV, 
	rHighLimit:=AHL 
);

END_FUNCTION_BLOCK

// oaksLibrary/Larm/fbLowLimitAlarm
// Larm låg gräns 
FUNCTION_BLOCK fbLowLimitAlarm EXTENDS fbAlarm
VAR_INPUT
	bEnable : BOOL; // FALSE = larm blockerat
	rProcessValue : REAL; // Ärvärde
	rLowLimit : REAL; // Larmgräns
END_VAR
VAR_OUTPUT
END_VAR
VAR
		iTemp3 : INT;
END_VAR

	SUPER^();
	bInput := rProcessValue < rLowLimit AND bEnable;

END_FUNCTION_BLOCK

// oaksLibrary/Larm/fbHighLimitAlarm
// Larm hög gräns 
FUNCTION_BLOCK fbHighLimitAlarm EXTENDS fbAlarm
VAR_INPUT
	bEnable : BOOL; // FALSE = larm blockerat
	rProcessValue : REAL; // Ärvärde
	rHighLimit : REAL; // Larmgräns
END_VAR
VAR_OUTPUT
END_VAR
VAR
		iTemp2 : INT;
END_VAR

	SUPER^();
	bInput := rProcessValue > rHighLimit AND bEnable;

END_FUNCTION_BLOCK

// oaksLibrary/Beräkning/fbHourDiff
// Beräknar förändring senaste timme
FUNCTION_BLOCK fbHourDiff
VAR_INPUT
	rTotalConsumedEnergy : REAL; //Totalt förbrukad energi
END_VAR
VAR_OUTPUT
	rEnergyConsumedEnergyDiff: REAL; //Förbrukad energi senaste timme
	rLastHourEnergyDiff: REAL; //Förbrukad energi föregående timme
END_VAR
VAR
	FB_BA_GetTime01 : tc2_ba.FB_BA_GetTime; 
	FB_BA_ExtTiSt01 : tc2_ba.FB_BA_ExtTiSt;
	wHour : WORD;
	fbHourTrig : R_TRIG;
	iTemp : INT;
	iCounter : INT;
END_VAR
VAR PERSISTENT
	wLastHourOfChange  : WORD;
	rTemporaryEnergy : REAL;
END_VAR

	FB_BA_GetTime01(bEn :=TRUE);	
	FB_BA_ExtTiSt01(stTi := FB_BA_GetTime01.stSysTi );

	IF FB_BA_ExtTiSt01.wHour <> wLastHourOfChange THEN
		fbHourTrig(CLK := TRUE);
	ELSE
		fbHourTrig(CLK := FALSE);
	END_IF
	
	IF fbHourTrig.Q THEN
		rLastHourEnergyDiff := rTotalConsumedEnergy - rTemporaryEnergy;
		rTemporaryEnergy := rTotalConsumedEnergy;
		wLastHourOfChange := FB_BA_ExtTiSt01.wHour;
	END_IF 

	rEnergyConsumedEnergyDiff := rTotalConsumedEnergy - rTemporaryEnergy;

END_FUNCTION_BLOCK

// oaksLibrary/Beräkning/fbMeanValueBC
// Beräknar medelvärde av samtliga värden i array som är inom inställda gränser BCLow och BCHigh. Arrayindex kan inte accessas som input till block där blocket utförs, utan måste accessas separat, t ex:
// fbMeanValueBC.InputArray[0] := VS01_GT11_PV;
// fbMeanValueBC.InputArray[1] := VS01_GT12_PV;
// [osv...]
// fbMeanValueBC(BCLow := 10.0, BCHigh := 100.0);

// Robert H, 2021-11-23
// Testat 2021-11-23

FUNCTION_BLOCK fbMeanValueBC
VAR_INPUT	
	InputArray	: ARRAY[0..99] OF REAL;		// Ingångsarray
	BCLow		: REAL;						// Lägsta tillåtna värde på ingång för beräkning
	BCHigh		: REAL;						// Högsta tillåtna värde på ingång för beräkning
END_VAR
VAR_OUTPUT
	MeanValue	: REAL;		// Beräknat medelvärde av tillåtna ingångsvärden
	BCValCnt	: INT;		// Antal tillåtna ingångsvärden i beräkning
END_VAR
VAR
	Index		: INT;
	InputSum	: REAL;
END_VAR

FOR Index := 0 TO 99 BY 1 DO
	
	IF (InputArray[Index] >= BCLow) AND (InputArray[Index] <= BCHigh) THEN
		BCValCnt := BCValCnt + 1;
		InputSum := InputSum + InputArray[Index];	
	END_IF;
	
	IF BCValCnt > 0 THEN
		MeanValue := InputSum / BCValCnt;
	END_IF;
	
END_FOR

BCValCnt := 0;
InputSum := 0;

END_FUNCTION_BLOCK

// oaksLibrary/Beräkning/fbOperatingHours
//OAKS AB
//2020-06-24
//Funktionsblock för beräkning av drifttid i timmar. Ingång för återställning av drifttid.
FUNCTION_BLOCK fbOperatingHours
VAR_INPUT
	bEnable : BOOL; //Aktiver drifttidsmätning
END_VAR

VAR_IN_OUT
	bReset : BOOL; //Nollställ drifttid
END_VAR
	
VAR_OUTPUT PERSISTENT
	rOperatingHours : UDINT := 0; //Drifttid
END_VAR

VAR
	FB_BA_GetTime01 : tc3_ba.FB_BA_GetTime; 
	FB_BA_ExtTiSt01 : tc3_ba.FB_BA_ExtTiSt;
	wLastMinOfChange: WORD;
	fbResetTon: TON;
END_VAR

VAR PERSISTENT
	rElapsedMin : REAL := 0; //Antal minuter i drift
END_VAR

	//Hämta klocka
	FB_BA_GetTime01(bEn :=TRUE);	
	FB_BA_ExtTiSt01(stTi := FB_BA_GetTime01.stSysTi );
		
	//Nollställ drifttid
	IF bReset THEN
		fbResetTon.IN := TRUE;
		IF fbResetTon.Q THEN
			bReset := FALSE;
			//Sätt drifttid och aktiva minuter till 0
			rOperatingHours := 0;
			rElapsedMin := 0;
		END_IF
	ELSE
		fbResetTon.IN := FALSE;
	END_IF
	fbResetTon.PT := T#5S;
	fbResetTon();
		
	//Om drifttidsmätning är aktiv och nuvarande minut ej överenstämmer med sparad minut ökas ökar driftid i minuter
	IF FB_BA_ExtTiSt01.wMinute <> wLastMinOfChange AND bEnable THEN
		wLastMinOfChange := FB_BA_ExtTiSt01.wMinute;
		rElapsedMin := rElapsedMin + 1;
	ELSE		
		rElapsedMin := rElapsedMin;
	END_IF
		
	//Om antalet minuter i drift överstiger eller är lika med 60 återställs timräkning och antal timmar räknas upp
	IF rElapsedMin >= 60 THEN
		rOperatingHours := rOperatingHours +1;
		rElapsedMin := 0;
	ELSE
		rOperatingHours := rOperatingHours;
		rElapsedMin := rElapsedMin;
	END_IF

END_FUNCTION_BLOCK

// oaksLibrary/Beräkning/fbScale6pSupTempRad
FUNCTION_BLOCK fbScale6pSupTempRad
VAR_INPUT
	 rX	 : ANY;	// Knyter man inget här används oaksGVL.rOutdoortemp som rX
END_VAR
VAR_OUTPUT
	 rY :	REAL;
END_VAR
VAR
 rTempUsed : REAL; // Uteluftstemperatur
 rXa : ARRAY[1..6] OF REAL;
 rYa : 	ARRAY[1..6] OF	REAL;
 rM :	REAL;	
 iI : 	INT;
END_VAR
VAR_INPUT PERSISTENT
	{attribute 'OPC.UA.DA' := '1'}
	Y1 AT %M* : REAL:=60;	//Utetemp/Börvärde~wp:[unit]°C[format]0.0
	{attribute 'OPC.UA.DA' := '1'}
	Y2 AT %M* :	REAL:=50;	//Utetemp/Börvärde~wp:[unit]°C[format]0.0
	{attribute 'OPC.UA.DA' := '1'}
	Y3 AT %M* :	REAL:=40;	//Utetemp/Börvärde~wp:[unit]°C[format]0.0
	{attribute 'OPC.UA.DA' := '1'}
	Y4 AT %M* :	REAL:=35;	//Utetemp/Börvärde~wp:[unit]°C[format]0.0
	{attribute 'OPC.UA.DA' := '1'}
	Y5 AT %M* :	REAL:=30;	//Utetemp/Börvärde~wp:[unit]°C[format]0.0
	{attribute 'OPC.UA.DA' := '1'}
	Y6 AT %M* :	REAL:=20;	//Utetemp/Börvärde~wp:[unit]°C[format]0.0
	{attribute 'OPC.UA.DA' := '1'}
	X1 AT %M* :	REAL:=-20;	//Utetemperatur~wp:[unit]°C[format]0.0
	{attribute 'OPC.UA.DA' := '1'}
	X2 AT %M* :	REAL:=-10;	//Utetemperatur~wp:[unit]°C[format]0.0
	{attribute 'OPC.UA.DA' := '1'}
	X3 AT %M* :	REAL:=0;	//Utetemperatur~wp:[unit]°C[format]0.0
	{attribute 'OPC.UA.DA' := '1'}
	X4 AT %M* :	REAL:=5;	//Utetemperatur~wp:[unit]°C[format]0.0
	{attribute 'OPC.UA.DA' := '1'}
	X5 AT %M* :	REAL:=10;	//Utetemperatur~wp:[unit]°C[format]0.0
	{attribute 'OPC.UA.DA' := '1'}
	X6 AT %M*:	REAL:=15;	//Utetemperatur~wp:[unit]°C[format]0.0
END_VAR

	//Temp select
	rTempUsed := F_GetTempToUse(rX);

//Breakpoints must be ascending
	IF (X2 <= X1) THEN X2 := X1 + 0.1; END_IF
	IF (X3 <= X2) THEN X3 := X2 + 0.1; END_IF
	IF (X4 <= X3) THEN X4 := X3 + 0.1; END_IF
	IF (X5 <= X4) THEN X5 := X4 + 0.1; END_IF
	IF (X6 <= X5) THEN X6 := X5 + 0.1; END_IF
 
	//Copy data to array
	rXa[1] := X1;
	rXa[2] := X2;
	rXa[3] := X3;
	rXa[4] := X4;
	rXa[5] := X5;
	rXa[6] := X6;
	rYa[1] := Y1;
	rYa[2] := Y2;
	rYa[3] := Y3;
	rYa[4] := Y4;
	rYa[5] := Y5;
	rYa[6] := Y6;

	//Calculate if value is out of boundaries	
	IF rTempUsed < rXa[1] THEN
		rY := rYa[1];
	END_IF;
	
	IF rTempUsed > rXa[6] THEN
		rY := rYa[6];
	END_IF;
		
	FOR iI := 1 TO 5 DO
		IF rTempUsed >= rXa[iI] AND rTempUsed <= rXa[iI + 1] THEN
			rM := (rYa[iI + 1] - rYa[iI])/(rXa[iI + 1]-rXa[iI]);
			rY := rYa[iI] + rM * (rTempUsed - rXa[iI]);
			EXIT;
		END_IF
	END_FOR

END_FUNCTION_BLOCK

// oaksLibrary/Datahantering/F_GetTempToUse
//Funktion för att välja vilken utetemperatur som ska användas. Knyter man ingenting väljs  oaksGVL.rOutdoorTemp. Knyter man en REAL väljs det värdet.
FUNCTION F_GetTempToUse : REAL
VAR_INPUT
	rTempToUse : ANY; //Temperatur för start/stopp. Om inget kopplas används oaksGVL.rOutdoorTemp
END_VAR
VAR
	pAnyReal : POINTER TO REAL;
END_VAR

//Temp select
IF rTempToUse.TypeClass = __SYSTEM.TYPE_CLASS.TYPE_REAL THEN
	pAnyReal := rTempToUse.pValue;
	F_GetTempToUse := pAnyReal^;
ELSE
	F_GetTempToUse := oaksGVL.rOutdoorTemp;
END_IF

END_FUNCTION

// oaksLibrary/Beräkning/fbScale6pSuptempVent
FUNCTION_BLOCK fbScale6pSuptempVent
VAR_INPUT
	 rX	 : ANY;	// Knyter man inget här används oaksGVL.rOutdoortemp som rX
END_VAR
VAR_OUTPUT
	 rY :	REAL;
END_VAR
VAR
 rTempUsed : REAL; // Uteluftstemperatur
 rXa : ARRAY[1..6] OF REAL;
 rYa : 	ARRAY[1..6] OF	REAL;
 rM :	REAL;	
 iI : 	INT;
END_VAR
VAR_INPUT PERSISTENT
	{attribute 'OPC.UA.DA' := '1'}
	Y1 AT %M* : REAL:=19;	//Utetemp/Börvärde~wp:[unit]°C[format]0.0
	{attribute 'OPC.UA.DA' := '1'}
	Y2 AT %M* :	REAL:=19;	//Utetemp/Börvärde~wp:[unit]°C[format]0.0
	{attribute 'OPC.UA.DA' := '1'}
	Y3 AT %M* :	REAL:=19;	//Utetemp/Börvärde~wp:[unit]°C[format]0.0
	{attribute 'OPC.UA.DA' := '1'}
	Y4 AT %M* :	REAL:=19;	//Utetemp/Börvärde~wp:[unit]°C[format]0.0
	{attribute 'OPC.UA.DA' := '1'}
	Y5 AT %M* :	REAL:=19;	//Utetemp/Börvärde~wp:[unit]°C[format]0.0
	{attribute 'OPC.UA.DA' := '1'}
	Y6 AT %M* :	REAL:=19;	//Utetemp/Börvärde~wp:[unit]°C[format]0.0
	{attribute 'OPC.UA.DA' := '1'}
	X1 AT %M* :	REAL:=-10;	//Utetemperatur~wp:[unit]°C[format]0.0
	{attribute 'OPC.UA.DA' := '1'}
	X2 AT %M* :	REAL:=-5;	//Utetemperatur~wp:[unit]°C[format]0.0
	{attribute 'OPC.UA.DA' := '1'}
	X3 AT %M* :	REAL:=0;	//Utetemperatur~wp:[unit]°C[format]0.0
	{attribute 'OPC.UA.DA' := '1'}
	X4 AT %M* :	REAL:=10;	//Utetemperatur~wp:[unit]°C[format]0.0
	{attribute 'OPC.UA.DA' := '1'}
	X5 AT %M* :	REAL:=20;	//Utetemperatur~wp:[unit]°C[format]0.0
	{attribute 'OPC.UA.DA' := '1'}
	X6 AT %M*:	REAL:=25;	//Utetemperatur~wp:[unit]°C[format]0.0
END_VAR

	//Temp select
	rTempUsed := F_GetTempToUse(rX);

//Breakpoints must be ascending
	IF (X2 <= X1) THEN X2 := X1 + 0.1; END_IF
	IF (X3 <= X2) THEN X3 := X2 + 0.1; END_IF
	IF (X4 <= X3) THEN X4 := X3 + 0.1; END_IF
	IF (X5 <= X4) THEN X5 := X4 + 0.1; END_IF
	IF (X6 <= X5) THEN X6 := X5 + 0.1; END_IF
 
	//Copy data to array
	rXa[1] := X1;
	rXa[2] := X2;
	rXa[3] := X3;
	rXa[4] := X4;
	rXa[5] := X5;
	rXa[6] := X6;
	rYa[1] := Y1;
	rYa[2] := Y2;
	rYa[3] := Y3;
	rYa[4] := Y4;
	rYa[5] := Y5;
	rYa[6] := Y6;

	//Calculate if value is out of boundaries	
	IF rTempUsed < rXa[1] THEN
		rY := rYa[1];
	END_IF;
	
	IF rTempUsed > rXa[6] THEN
		rY := rYa[6];
	END_IF;
		
	FOR iI := 1 TO 5 DO
		IF rTempUsed >= rXa[iI] AND rTempUsed <= rXa[iI + 1] THEN
			rM := (rYa[iI + 1] - rYa[iI])/(rXa[iI + 1]-rXa[iI]);
			rY := rYa[iI] + rM * (rTempUsed - rXa[iI]);
			EXIT;
		END_IF
	END_FOR

END_FUNCTION_BLOCK

// oaksLibrary/Beräkning/fbSfpCalc
//OAKS AB 2023-02-08 Ver. b0.1
//Funktionsblock för SFP beräkning.
FUNCTION_BLOCK fbSfpCalc 

VAR
	rSfpGf					: REAL;
	rSfpTf					: REAL;
	rSfpFf					: REAL;
END_VAR

VAR_INPUT
	bEnable	AT %M* : BOOL := TRUE;
	rFlowSupply AT %M* : REAL; //Flöde tilluft~wp:[unit]m3/s[trendoptions]i:300
	rFlowExhaust AT %M* : REAL; //Flöde frånluft~wp:[unit]m3/s[trendoptions]i:300
	rEffectSupply AT %M* : REAL; //Effekt tilluft~wp:[unit]kW[trendoptions]i:300
	rEffectExhaust AT %M* : REAL; //Effekt frånluft~wp:[unit]kW[trendoptions]i:300
END_VAR

VAR_OUTPUT
	rSFP AT %M* : REAL; //SFP-beräkning~wp:[unit]kW/(m3/s)[format]0.0
END_VAR

VAR_INPUT PERSISTENT

END_VAR


IF bEnable THEN
	rSfpGf := MAX(rFlowSupply, rFlowExhaust);
	rSfpTf := ABS(rEffectSupply);
	rSfpFf := ABS(rEffectExhaust);
	
	IF rSfpGf <> 0 AND rSfpTf <> 0 AND rSfpFf <> 0 THEN
		rSFP := ABS((rSfpTf + rSfpFf)/rSfpGf);
	ELSE
		rSFP := 0.0;		
	END_IF
ELSE
	rSFP := 0.0;
END_IF

END_FUNCTION_BLOCK

// oaksLibrary/Beräkning/fbSunClock
//Block för beräkning av soluppgång och solnedgång. 
//Räknar ut tid för soluppgång och solnedgång baserat på inställd Latitude och Longitude. Belysningsvillkorets aktivering och avaktivering går att förskjuta med inställd tid.
FUNCTION_BLOCK fbSunClock
VAR PERSISTENT
	{attribute 'OPC.UA.DA' := '1'}
	SP1 AT %M* : REAL := 57.7089;//Latitude (-90 till 90)~wp:[format]0.000000
	{attribute 'OPC.UA.DA' := '1'}
	SP2 AT %M* : REAL := 11.9746;//Longitude (-180 to 180)~wp:[format]0.000000
	{attribute 'OPC.UA.DA' := '1'}
	SP3 AT %M* : INT := 30; //Senarelägg avakt. av bel.villkor med ins. tid~wp:[unit]min[format]0
	{attribute 'OPC.UA.DA' := '1'}
	SP4 AT %M* : INT := 30; //Tidigarelägg akt. av bel.villkor med ins. tid~wp:[unit]min[format]0
END_VAR
VAR_OUTPUT
	V AT %M*  : BOOL;//Driftvillkor belysning~wp:[trendoptions]i:14400, t:1
END_VAR
VAR
	sSoluppgangForskjuten : STRING;	
	sSolnedgangForskjuten : STRING;	

	dIntSunRiseForskjutning : DINT;
	dIntSunSetForskjutning : DINT;
	
	todRiseForskjutning : TOD;
	todSunSetForskjutning : TOD;
	
	iSunRiseForskjutning : INT;
	iSunSetForskjutning : INT;

	itemp : int;
	fbToFTidsFordrojningDriftvillkor : TOF;
	
	fbGetTimeZoneInformation01 : FB_GetTimeZoneInformation;
	ST_TimeZoneInformation01  : ST_TimeZoneInformation;	
	diSommarVinterTidsForskjutning : DINT; 

	rLatitude AT %M* : REAL := 57.7089;//Latitude 
	rLongitude AT %M* : REAL := 11.9746;//Longitude
	(*
		Göteborg: 
		<br>Latitude = 57.7089 
		<br>Longitude = 11.9746 
		<br>Stockholm: 
		<br>Latitude = 59.3293 
		<br>Longitude = 18.0686 
		<br>Malmö: 
		<br>Latitude = 55.6050 
		<br>Longitude = 13.0038
		<br>Jokkmokk: 
		<br>Latitude = 66.6070 
		<br>Longitude = 19.8229
		<br>
		<br>För att hitta andra städers koordinater googla "Vilka koordinater har STAD?~wp:"
	*)
	PV4 AT %M* : STRING := ' ';
	{attribute 'OPC.UA.DA' := '1'}
	PV AT %M* : STRING := ' '; //Soluppgång och solnedgång~wp:
	{attribute 'OPC.UA.DA' := '1'}
	PV1 AT %M* : STRING := ' '; //Belysningsvillkor till och från~wp:
	{attribute 'OPC.UA.DA' := '1'}
	PV6 AT %M* : INT; //Soluppgång~wp:[format]00:00[engmin]0[engmax]2400
	{attribute 'OPC.UA.DA' := '1'}
	PV7 AT %M* : INT; //Solnedgång~wp:[format]00:00[engmin]0[engmax]2400
	{attribute 'OPC.UA.DA' := '1'}
	PV8 AT %M* : STRING := ' '; //Räknar ut tid för soluppgång och solnedgång baserat på inställd Latitude och Longitude. Belysningsvillkorets aktivering och avaktivering går att förskjuta med inställd tid.~wp:
	bInnanSoluppgang : BOOL;
	bEfterSolnedgang : BOOL;
	sSolnedgang : STRING;	
	sSoluppgang : STRING;	
	sSun_setString : STRING;	
	sSun_riseString : STRING;	
	iStringLength : INT;
	MIDDAY : TOD;			(*	astrological midday in hours when sun stands at south direction	*)
	SUN_RISE : TOD;				(*	sun rise for current day in local time *)
	SUN_SET : TOD;				(*	sun set for current day in local time *)
	SUN_DECLINATION : REAL;		(*	sun declination above horizon at midday in degrees	*)	
	H : REAL := -0.83333333333;	(* heighth above horizon for sunrise *)
	PI2 : REAL := 	6.28318530717958647692528676655900576;	(* PI * 2 *)
	UTC : DATE;	
	fbToggle01 : fbToggle;
	fbLocalSysTime  : FB_LocalSystemTime;
	stSysTime01  : TIMESTRUCT;
	tTimeInDateAndTime  : DT;	
	tTimeInDate : DATE;
	date1 : DATE;	
	FB_BA_GetTime01 : tc2_ba.FB_BA_GetTime; 
	FB_BA_ExtTiSt01 : tc2_ba.FB_BA_ExtTiSt;
	dk: REAL;						(* sun declination at midday *)
	delta: TIME;					(* delta from midday for sunrise and sunset  *)
	b: REAL;
	rSunRiseInt : REAL; 
	tTestTOD : TOD;
	iSunrise : INT;
	iSunset : INT;
	
END_VAR
VAR
	bUpdate : BOOL := true;	

	DayMinutes:REAL; //Dagsljus i minuter
	RiseMinutes:REAL; //Soluppgångstid i minuter
	NowMinutes:REAL; //Nu i minuter
	PassedMinutes:REAL; //Minuter som har passerat sen soluppgång
	PERCENT_PV AT %M* :REAL; //Del av dag som passerat~wp:[unit]%[format]0
	DayStruct: OTSTRUCT; //Struct för dagsljus-tid
	RiseStruct: OTSTRUCT; //Struct för soluppgongs-tid
	SetStruct: OTSTRUCT; //Struct för Solnedgångstid
END_VAR
(*
version 1.7	25. jan. 2011
programmer 	hugo
tested by	tobias

this FUNCTION block calculates the sun rise, sun set, sun offset at midday sun declination for a given date 
for performance reasons the algorithm has been simplified and is accurate within a few minutes only 
the times are calculated in utc and have to be corrected for the given time zone
this correction is not done within sun_time because it would be a problem on days where dst is enabled or disabled

*)

	mPercentageOfDay();

	IF 	SP1 > 90 THEN
		SP1 := 90; 
	ELSIF SP1 < -90 THEN
		SP1 := -90;
	END_IF
	
	IF SP1 <= 90 AND SP1 >= -90 THEN
		rLatitude := SP1; 
	END_IF

	IF 	SP2 > 180 THEN
		SP2 := 180; 
	ELSIF SP2 < -180 THEN
		SP2 := -180;
	END_IF

	IF SP2 <= 180 AND SP2 >= -180 THEN
		rLongitude := SP2; 
	END_IF
	


	IF SP3 < 0 THEN
		SP3 := 0;
	ELSIF SP3 > 360 THEN
		SP3 := 360;
	END_IF;
	
	IF SP4 < 0 THEN
		SP4 := 0;
	ELSIF SP4 > 360 THEN 
		SP4 := 360;
	END_IF
	// HÄmta tid
	fbToggle01(bStart:=TRUE , tTimeOn:=T#10S , tTimeOff:= T#10S, bOutput=> );
	fbLocalSysTime(
	sNetID:= , 
	bEnable:= fbToggle01.bOutput, 
	dwCycle:= , 
	dwOpt:= , 
	tTimeout:= , 
	bValid=> , 
	systemTime=> stSysTime01, 
	tzID=> );
	tTimeInDateAndTime := SYSTEMTIME_TO_DT(stSysTime01);
	UTC := DT_TO_DATE (tTimeInDateAndTime);
	
	// Kollar om det är sommar eller vintertid
	fbGetTimeZoneInformation01(
	sNetID:= , 
	bExecute:=fbtoggle01.bOutput , 
	tTimeout:= , 
	bBusy=> , 
	bError=> , 
	nErrID=> , 
	tzID=> , 
	tzInfo=> ST_TimeZoneInformation01);
	IF fbLocalSysTime.tzID = E_TimeZoneID.eTimeZoneID_Daylight THEN 
		diSommarVinterTidsForskjutning := 120*60000; // Aktuell tidsförskjutning sommar och vintertid
	ELSE
		diSommarVinterTidsForskjutning := 60*60000;
	END_IF;
	// Uträkning
	B := rLatitude * 0.0174532925199433;
	MIDDAY := SUN_MIDDAY(rLongitude, utc);
	DK := 0.40954 * SIN(0.0172 * (INT_TO_REAL(DAY_OF_YEAR(utc)) - 79.35));
	sun_declination := DEG(DK);
	IF sun_declination > 180.0 THEN sun_declination := sun_declination - 360.0; END_IF;
	sun_declination := 90.0 - rLatitude + sun_declination;
	delta := HOUR_TO_TIME(ACOS((SIN(RAD(H)) - SIN(B) * SIN(DK)) / (COS(B) * COS(DK))) * 3.819718632);
	sun_rise := MIDDAY - delta + DINT_TO_TIME(diSommarVinterTidsForskjutning);
	sun_set := MIDDAY + delta + DINT_TO_TIME(diSommarVinterTidsForskjutning);

	// Soluppgång
	iStringLength := LEN(TOD_TO_STRING(sun_rise)) - 4;
	sSun_riseString := RIGHT(TOD_TO_STRING(sun_rise),iStringLength); 
	sSoluppgang := CONCAT('Soluppgång: ', sSun_riseString);
	iSunrise := HOUR(sun_rise)*100+MINUTE(sun_rise);
	PV6 := iSunrise; // För trendning i webport
	// Solnedgång
	iStringLength := LEN(TOD_TO_STRING(sun_set)) - 4;
	sSun_setString := RIGHT(TOD_TO_STRING(sun_set),iStringLength); 
	sSolnedgang := CONCAT('Solnedgång: ', sSun_setString);
	iSunset := HOUR(sun_set)*100+MINUTE(sun_set);
	PV7 := iSunset; // För trendning i webport
	
	dIntSunRiseForskjutning :=  SP3;
	
	todRiseForskjutning := sun_rise + DINT_TO_TIME(dIntSunRiseForskjutning*60000);
	iSunRiseForskjutning := HOUR(todRiseForskjutning)*100+MINUTE(todRiseForskjutning);
	bInnanSoluppgang :=  oaksgvl.iHourAndMinute < iSunRiseForskjutning;

	dIntSunSetForskjutning :=  SP4;
	todSunSetForskjutning := sun_set - DINT_TO_TIME(dIntSunSetForskjutning*60000);
	iSunSetForskjutning := HOUR(todSunSetForskjutning)*100+MINUTE(todSunSetForskjutning);
	bEfterSolnedgang :=  oaksgvl.iHourAndMinute >  iSunSetForskjutning;
	
	fbToFTidsFordrojningDriftvillkor(IN:=bInnanSoluppgang OR bEfterSolnedgang , PT:= T#5S, Q=> , ET=> );
	
	V := fbToFTidsFordrojningDriftvillkor.Q;
	
	PV := mSoluppgangOchSolnedgang(sSoluppgang, sSolnedgang);
	
	
	iStringLength := LEN(TOD_TO_STRING(todRiseForskjutning)) - 4;
	sSoluppgangForskjuten  := RIGHT(TOD_TO_STRING(todRiseForskjutning),iStringLength); 
	
	iStringLength := LEN(TOD_TO_STRING(todSunSetForskjutning)) - 4;
	sSolnedgangForskjuten  := RIGHT(TOD_TO_STRING(todSunSetForskjutning),iStringLength); 
	
	
	PV1 := mSolnedOchUppGangForskjuten(sSoluppgangForskjuten,sSolnedgangForskjuten);
(* revision history

rev 1.1	hm	20.1.2007
	deleted unused variables sun_riseR and sun_setR

rev 1.2 hm 17.4.2007
	corrected error while sun:midday would not be corrected for longitude.

rev 1.3	hm	6. jan 2008
	performance improvements

rev	1.4 hm	17. jan 2008
	calculation is now only performed once a day

hm	10. mar. 2009	rev 1.5
	improved performance
	calculation will be performed on every call to allow movong installations

hm	26. jul 2009	rev 1.6
	fixed a problem with wrong midday calculation

hm	25. jan. 2011	rev 1.7
	using function sun_midday
	corrected angle of sun_declination
	added input H
*)

METHOD PRIVATE DAY_OF_YEAR : INT
VAR_INPUT
	IDATE : DATE;
END_VAR


(*
version 1.4		28. jan. 2011
programmer 	hugo
tested by		oscat

calculates the day of the year

*)
DAY_OF_YEAR := UDINT_TO_INT((DATE_TO_UDINT(idate) / UDINT#86400) MOD UDINT#1461);
IF DAY_OF_YEAR > 729 THEN
	IF DAY_OF_YEAR > 1095 THEN DAY_OF_YEAR := DAY_OF_YEAR - 1095; ELSE DAY_OF_YEAR := DAY_OF_YEAR - 729; END_IF;
ELSIF DAY_OF_YEAR > 364 THEN
	DAY_OF_YEAR := DAY_OF_YEAR - 364;
ELSE
	DAY_OF_YEAR := DAY_OF_YEAR + 1;
END_IF;


(*
DAY_OF_YEAR := DWORD_TO_INT((DATE_TO_DWORD(idate) - DATE_TO_DWORD(YEAR_BEGIN(YEAR_OF_DATE(idate)))) / 86400) + 1;
*)


(* revivision history
hm	4. aug. 2007		rev 1.0
	original version

hm	1. oct. 2007		rev 1.1
	added compatibility to STEP7

hm	4. jan. 2008		rev 1.2
	changed code for better performance

hm	7. oct. 2008		rev 1.3
	changed name of function year to year_of_date

hm	28. jan. 2011	rev 1.4
	improved code
*)
END_METHOD

METHOD PRIVATE DEG : REAL
VAR_INPUT
	rad : REAL;
END_VAR


(*
version 1.2	10. mar. 2009
programmer 	hugo
tested by		tobias

this function converts degrees into Radiant
execution time on wago 750 - 841 =  10  us
*)
DEG := MODR(57.29577951308232 * RAD, 360.0);

(* revision history
hm	4. aug 2006	rev 1.0
	original version

hm 16. oct 2007	rev 1.1
	added modr statement which prohibits deg to become bigger than 360

hm	10. mar. 2009	rev 1.2
	real constants updated to new systax using dot
*)
END_METHOD

METHOD PRIVATE FLOOR2 : DINT
VAR_INPUT
	X : REAL;
END_VAR



(*
version 1.1	4. apr. 2008
programmer 	hugo
tested by		tobias

This is a rounding function which returns the biggest possible integer which is less or equal to X.
floor2(3.14) = 3
floor2(-3.14) = -4

*)
FLOOR2 := REAL_TO_DINT(X);
IF DINT_TO_REAL(FLOOR2) > X THEN
	FLOOR2 := FLOOR2 - 1;
END_IF;

(* revision history
hm	21. mar. 2008	rev 1.0
	originlal version

hm	4. apr. 2008	rev 1.1
	added type conversion to avoid warnings under codesys 3.0
*)
END_METHOD

METHOD PRIVATE HOUR : INT
VAR_INPUT
	itod : TOD;
END_VAR


(*
version 1.1	2 okt 2006
programmer 	hugo
tested by	tobias

extracts the hour of a Time_of_day 
*)
HOUR := DWORD_TO_INT(TOD_TO_DWORD(itod) / 3600000);


(* change history
hm 4. aug 2006	rev 1.0
	original version

hm 2.10.2006 	rev 1.1
	changed name of input to itod

*)
END_METHOD

METHOD PRIVATE HOUR_TO_TIME : TIME
VAR_INPUT
	IN : REAL;
END_VAR


(*
version 1.2	24. feb. 2009
programmer 	hugo
tested by		tobias

converts an amount of hours in real to time

*)
HOUR_TO_TIME := DWORD_TO_TIME(REAL_TO_DWORD(IN * 3600000));


(* revision history
hm		4. aug 2006	rev 1.0
	original version

hm	14. mar. 2008	rev 1.1
	rounded the input after the last digit

hm	24. feb. 2009	rev 1.2
	changed input to IN
*)
END_METHOD

METHOD PRIVATE HOUR_TO_TOD : TOD
VAR_INPUT
	IN : REAL;
END_VAR


(*
version 1.2	24. feb 2009
programmer 	hugo
tested by		tobias

converts an amount of hours in real to time of day TOD.

*)
HOUR_TO_TOD := DWORD_TO_TOD(REAL_TO_DWORD(IN * 3600000));


(* revision history
hm	4. aug. 2006	rev 1.0
	original version

hm	14. mar. 2008	rev 1.1
	rounded the input after the last digit

hm	24. feb. 2009	rev 1.2
	changed input to IN
*)
END_METHOD

METHOD PRIVATE MINUTE : INT
VAR_INPUT
	itod : TOD;
END_VAR


(*
version 1.1	2 oct 2006
programmer 	hugo
tested by	tobias

extracts the minutes out of TOD truncating the seconds 

*)
MINUTE := DWORD_TO_INT(TOD_TO_DWORD(itod) / 60000 - TOD_TO_DWORD(itod) / 3600000 * 60);


(* change history

2.10.2006 changes name of input to itod

*)
END_METHOD

METHOD PROTECTED MODR : REAL
VAR_INPUT
	IN : REAL;
	DIVI : REAL;
END_VAR


(*
version 1.5	10. mar. 2009
programmer 	hugo
tested by		tobias

this is a modulo funtion for real numbers
modr(5.5,2.5) = 0.5

*)
IF divi = 0.0 THEN
	MODR := 0.0;
ELSE
	MODR := in - DINT_TO_REAL(FLOOR2(in / divi)) * divi;
END_IF;

(* revision history

hm	4. aug.2006		rev 1.0

hm	28. jan.2007	rev 1.1
	modr(x,0) will deliver the result 0

hm	21. mar 2008	rev 1.2
	use D_trunc for compatibility reasons

hm	4. apr. 2008	rev 1.3
	added type conversion to avoid warnings under codesys 3.0

hm	31. oct. 2008	rev 1.4
	changed algorithm to the more common version using floor instead of TRUNC

hm	10. mar. 2009	rev 1.5
	real constants updated to new systax using dot

*)
END_METHOD

METHOD PRIVATE mPercentageOfDay
VAR_INPUT
END_VAR
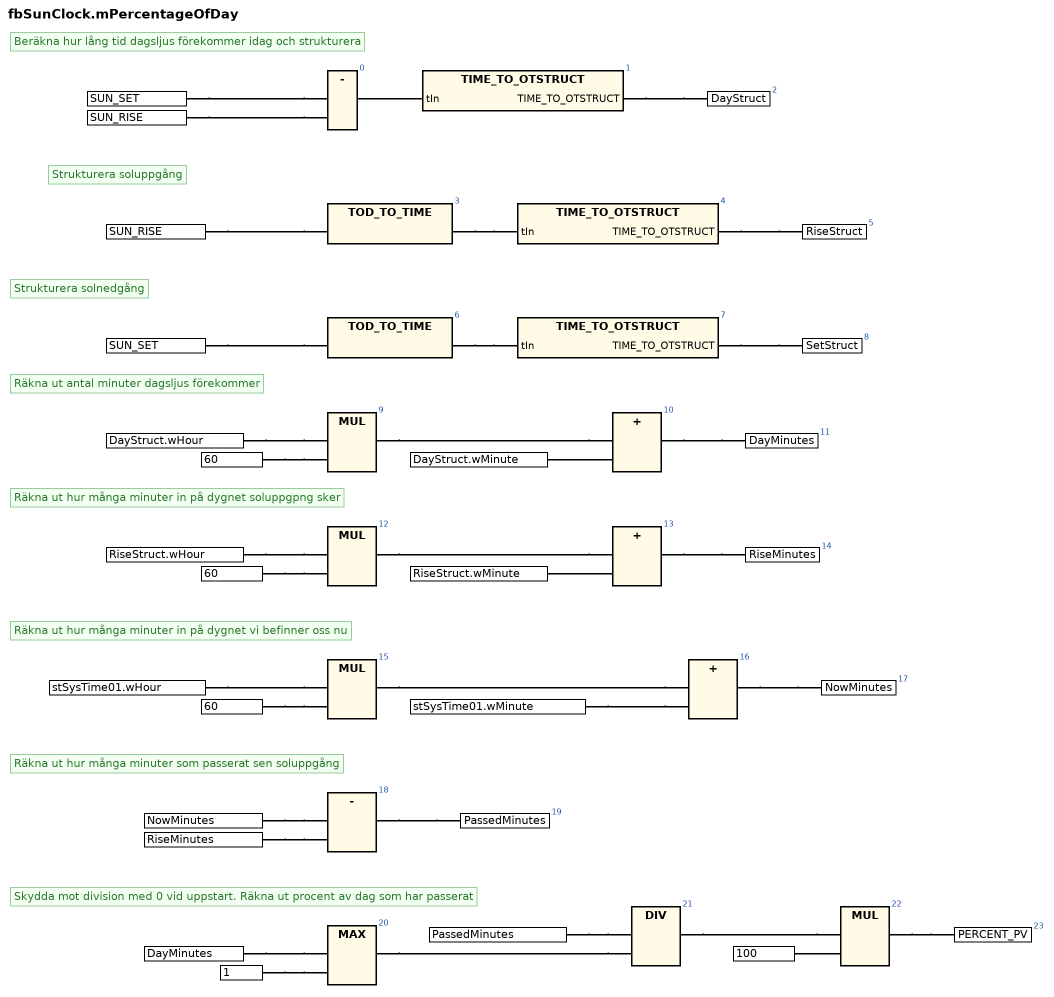
// Beräkna hur lång tid dagsljus förekommer idag och strukturera
DayStruct := TIME_TO_OTSTRUCT(tIn := SUN_SET - SUN_RISE);
// Strukturera soluppgång
RiseStruct := TIME_TO_OTSTRUCT(tIn := TOD_TO_TIME(SUN_RISE));
// Strukturera solnedgång
SetStruct := TIME_TO_OTSTRUCT(tIn := TOD_TO_TIME(SUN_SET));
// Räkna ut antal minuter dagsljus förekommer
DayMinutes := DayStruct.wHour * 60 + DayStruct.wMinute;
// Räkna ut hur många minuter in på dygnet soluppgpng sker
RiseMinutes := RiseStruct.wHour * 60 + RiseStruct.wMinute;
// Räkna ut hur många minuter in på dygnet vi befinner oss nu
NowMinutes := stSysTime01.wHour * 60 + stSysTime01.wMinute;
// Räkna ut hur många minuter som passerat sen soluppgång
PassedMinutes := NowMinutes - RiseMinutes;
// Skydda mot division med 0 vid uppstart. Räkna ut procent av dag som har passerat
PERCENT_PV := (PassedMinutes / MAX(DayMinutes, 1)) * 100;
END_METHOD

METHOD PRIVATE mSolnedOchUppGangForskjuten : STRING
VAR_INPUT
	sSoluppgang : STRING;	
	sSolnedgang : STRING;	
END_VAR
VAR 
	sTemp : STRING;
	
	sSoluppgangMedStrang : STRING;	
	sSolnedgangMedStrang : STRING;	
END_VAR
sSoluppgangMedStrang := CONCAT('Belysningsvillkor från: ',sSoluppgang);
sSolnedgangMedStrang := CONCAT('Belysningsvillkor till: ',sSolnedgang);


sTemp := CONCAT(sSoluppgangMedStrang, ' , '); 
mSolnedOchUppGangForskjuten := CONCAT(sTemp, sSolnedgangMedStrang);
END_METHOD

METHOD PRIVATE mSoluppgangOchSolnedgang : STRING
VAR_INPUT
	sSoluppgang : STRING;	
	sSolnedgang : STRING;	
END_VAR
VAR 
	sTemp : STRING;
END_VAR
sTemp := CONCAT(sSoluppgang, ' , '); 
mSoluppgangOchSolnedgang := CONCAT(sTemp, sSolnedgang);
END_METHOD

METHOD PRIVATE RAD : REAL
VAR_INPUT
	deg : REAL;
END_VAR


(*
version 1.2	18. oct. 2008
programmer 	hugo
tested by	tobias

this function converts Radiant to degrees

*)
RAD := MODR(0.0174532925199433 * DEG, PI2); // skapade PI2 lokalt i blocket istället för att slippa kopiera med CONSTANTS_MATH från OSCAT BASIC.
//RAD := MODR(0.0174532925199433 * DEG, math.PI2);

(* revision history
hm	4. aug 2006		rev 1.0
	original version

hm 	16. oct 2007	rev 1.1
	added modr statement which prohibits rad to become bigger than 2PI

hm	18. oct 2008	rev 1.2
	using math constants

*)
END_METHOD

METHOD PRIVATE SUN_MIDDAY : TOD
VAR_INPUT
	LON : REAL;
	UTC : DATE;
END_VAR
VAR
	T : REAL;
	OFFSET : REAL;
END_VAR

(*
version 1.0	26. jan. 2011
programmer 	hugo
tested by	oscat

this FUNCTION calculates the time when the sun stand exactly south of a given location.

*)
T := INT_TO_REAL(DAY_OF_YEAR(utc));
OFFSET := -0.1752 * SIN(0.033430 * T + 0.5474) - 0.1340 * SIN(0.018234 * T - 0.1939);
SUN_MIDDAY := HOUR_TO_TOD(12.0 - OFFSET - lon * 0.0666666666666);


(* revision history

hm	26. jan. 2011	rev 1.0
	initial release

*)
END_METHOD

END_FUNCTION_BLOCK

// oaksLibrary/fbToggle
// Toggle-funktion. Togglar bOutput med inställd intervall när bStart är till.
FUNCTION_BLOCK fbToggle
VAR_INPUT
	bStart : BOOL;
	tTimeOn : TIME := T#10S;
	tTimeOff : TIME := T#10S;
END_VAR
VAR_OUTPUT
	bOutput : BOOL;
END_VAR
VAR
	fbTrigger : r_trig;
	fbTon1 : ton;
	fbTof2 : tof;
END_VAR

IF bStart THEN
	fbTon1(IN:= NOT fbTof2.Q, PT:= tTimeOn , Q=> , ET=> );
	IF fbTon1.Q THEN
		fbTrigger(CLK:=TRUE , Q=> );
		fbTof2(IN:=fbTrigger.Q , PT:=tTimeOff , Q=> , ET=> );
	ELSE
		fbTof2(IN:=FALSE , PT:=tTimeOff , Q=> , ET=> );
		fbTrigger(CLK:=FALSE , Q=> );		
	END_IF
	bOutput := fbTof2.Q;
ELSE
	bOutput := FALSE;
END_IF
fbTof2();
fbTon1();

END_FUNCTION_BLOCK

// oaksLibrary/Beräkning/fCalcFlow
//Allmän flödesberäkning genom tryck och K-faktor
FUNCTION fCalcFlow : REAL
VAR_INPUT
	bFan : BOOL; //Fläktindikering för att tillåta uträkningen
	rPa : REAL; //Tryckvärde
	rKfaktor : REAL; //K-faktor
END_VAR

IF bFan AND rPa > 0.1 AND rKfaktor > 0.1 THEN
	//fCalcFlow:= ((1/rKfaktor) * (SQRT(rPa)))*1000;
	fCalcFlow:= ((rKfaktor * (SQRT(rPa)))/3.6);
ELSE
	fCalcFlow := 0;
END_IF

END_FUNCTION

// oaksLibrary/Beräkning/fCalcFlowfbNicotraGerbhardtRLM
//Beräkna flöde från tryck för Nicotra Gerbhardt RLM
FUNCTION fCalcFlowfbNicotraGerbhardtRLM : REAL
VAR_INPUT
	bFan : BOOL; //Fläktindikering för att tillåta uträkningen
	rPa : REAL; //Tryckvärde
	rKfaktor : REAL; //K-faktor
END_VAR

IF bFan AND rPa > 0.1 AND rKfaktor > 0.1 THEN
	//fCalcFlow:= ((1/rKfaktor) * (SQRT(rPa)))*1000;
	fCalcFlowfbNicotraGerbhardtRLM:= ((rKfaktor * (SQRT((2/1.29) * rPa)))/3.6);
ELSE
	fCalcFlowfbNicotraGerbhardtRLM := 0;
END_IF

END_FUNCTION

// oaksLibrary/Beräkning/fScale12pInternalSetpoint
// Skalar om x till y med 12 punkter. Exempelvis för utekompensering. Ingen VAR-IN-OUT.
FUNCTION fScale12pInternalSetpoint : REAL
VAR_INPUT
	 rX	 : ANY;
	 y1 : 	REAL;	
	 y2:	REAL;	
	 y3:	REAL;	
	 y4:	REAL;	
	 y5:	REAL;	
	 y6:	REAL;
	 y7: 	REAL;	
	 y8:	REAL;	
	 y9:	REAL;	
	 y10:	REAL;	
	 y11:	REAL;	
	 y12:	REAL;
	 x1:	REAL;	
	 x2:	REAL;	
	 x3:	REAL;	
	 x4:	REAL;	
	 x5:	REAL;	
	 x6:	REAL;
	 x7:	REAL;	
	 x8:	REAL;	
	 x9:	REAL;	
	 x10:	REAL;	
	 x11:	REAL;	
	 x12:	REAL;	
END_VAR
VAR
	 rTempUsed : REAL; // Uteluftstemperatur
	 rXa : ARRAY[1..12] OF REAL;
	 rYa : 	ARRAY[1..12] OF	REAL;
	 rM :	REAL;	
	 iI : 	INT;
END_VAR

//Temp select
	rTempUsed := F_GetTempToUse(rX);
	
//Breakpoints must be ascending
	IF (x2 <= x1) THEN x2 := x1 + 0.1; END_IF
	IF (x3 <= x2) THEN x3 := x2 + 0.1; END_IF
	IF (x4 <= x3) THEN x4 := x3 + 0.1; END_IF
	IF (x5 <= x4) THEN x5 := x4 + 0.1; END_IF
	IF (x6 <= x5) THEN x6 := x5 + 0.1; END_IF
	
	IF (x7 <= x6) THEN x7 := x6 + 0.1; END_IF
	IF (x8 <= x7) THEN x8 := x7 + 0.1; END_IF
	IF (x9 <= x8) THEN x9 := x8 + 0.1; END_IF
	IF (x10 <= x9) THEN x10 := x9 + 0.1; END_IF
	IF (x11 <= x10) THEN x11 := x10 + 0.1; END_IF
	IF (x12 <= x11) THEN x12 := x11 + 0.1; END_IF
 
	//Copy data to array
	rXa[1] := x1;
	rXa[2] := x2;
	rXa[3] := x3;
	rXa[4] := x4;
	rXa[5] := x5;
	rXa[6] := x6;
	rXa[7] := x7;
	rXa[8] := x8;
	rXa[9] := x9;
	rXa[10] := x10;
	rXa[11] := x11;
	rXa[12] := x12;
		
	rYa[1] := y1;
	rYa[2] := y2;
	rYa[3] := y3;
	rYa[4] := y4;
	rYa[5] := y5;
	rYa[6] := y6;
	rYa[7] := y7;
	rYa[8] := y8;
	rYa[9] := y9;
	rYa[10] := y10;
	rYa[11] := y11;
	rYa[12] := y12;

	//Calculate if value is out of boundaries	
	IF rTempUsed < rXa[1] THEN
		fScale12pInternalSetpoint := rYa[1];
	ELSIF rTempUsed > rXa[12] THEN
		fScale12pInternalSetpoint := rYa[12];
	ELSE	
		FOR iI := 1 TO 11 DO
			IF rTempUsed >= rXa[iI] AND rTempUsed <= rXa[iI + 1] THEN
				rM := (rYa[iI + 1] - rYa[iI])/(rXa[iI + 1]-rXa[iI]);
				fScale12pInternalSetpoint := rYa[iI] + rM * (rTempUsed - rXa[iI]);
				EXIT;
			END_IF
		END_FOR
	END_IF;

END_FUNCTION

// oaksLibrary/Beräkning/fScale20p
// Skalar om x till y med 20 punkter.
FUNCTION fScale20p : REAL
VAR_INPUT
	 rX	 : ANY;	// Knyter man inget här används oaksGVL.rOutdoortemp som rX	
END_VAR
VAR_IN_OUT
	 Y1 : 	REAL;	
	 Y2:	REAL;	
	 Y3:	REAL;	
	 Y4:	REAL;	
	 Y5:	REAL;	
	 Y6:	REAL;	
	 Y7:	REAL;	
	 Y8 : 	REAL;	
	 Y9:	REAL;	
	 Y10:	REAL;	
	 Y11:	REAL;	
	 Y12:	REAL;	
	 Y13:	REAL;	
	 Y14:	REAL;
	 Y15:	REAL;
	 Y16:	REAL;
	 Y17:	REAL;
	 Y18:	REAL;
	 Y19:	REAL;
	 Y20:	REAL;
	 X1:	REAL;	
	 X2:	REAL;	
	 X3:	REAL;	
	 X4:	REAL;	
	 X5:	REAL;	
	 X6:	REAL;	
	 X7:	REAL;
	 X8:	REAL;
	 X9:	REAL;
	 X10:	REAL;
	 X11:	REAL;
	 X12:	REAL;
	 X13:	REAL;
	 X14:	REAL;
	 X15:	REAL;
	 X16:	REAL;
	 X17:	REAL;
	 X18:	REAL;
	 X19:	REAL;
	 X20:	REAL;	
END_VAR
VAR
	 rTempUsed : REAL;
	 rXa : ARRAY[1..20] OF REAL;
	 rYa : 	ARRAY[1..20] OF	REAL;
	 rM :	REAL;	
	 iI : 	INT;
END_VAR

//Temp select
	rTempUsed := F_GetTempToUse(rX);

//Breakpoints must be ascending
	IF (X2 <= X1) THEN X2 := X1 + 0.1; END_IF
	IF (X3 <= X2) THEN X3 := X2 + 0.1; END_IF
	IF (X4 <= X3) THEN X4 := X3 + 0.1; END_IF
	IF (X5 <= X4) THEN X5 := X4 + 0.1; END_IF
	IF (X6 <= X5) THEN X6 := X5 + 0.1; END_IF
	IF (X7 <= X6) THEN X7 := X6 + 0.1; END_IF
	IF (X8 <= X7) THEN X8 := X7 + 0.1; END_IF
	IF (X9 <= X8) THEN X9 := X8 + 0.1; END_IF
	IF (X10 <= X9) THEN X10 := X9 + 0.1; END_IF
	IF (X11 <= X10) THEN X11 := X10 + 0.1; END_IF
	IF (X12 <= X11) THEN X12 := X11 + 0.1; END_IF
	IF (X13 <= X12) THEN X13 := X12 + 0.1; END_IF
	IF (X14 <= X13) THEN X14 := X13 + 0.1; END_IF
	IF (X15 <= X14) THEN X15 := X14 + 0.1; END_IF
	
	IF (X16 <= X15) THEN X16 := X15 + 0.1; END_IF
	IF (X17 <= X16) THEN X17 := X16 + 0.1; END_IF
	IF (X18 <= X17) THEN X18 := X17 + 0.1; END_IF
	IF (X19 <= X18) THEN X19 := X18 + 0.1; END_IF
	IF (X20 <= X19) THEN X20 := X19 + 0.1; END_IF
 
	//Copy data to array
	rXa[1] := X1;
	rXa[2] := X2;
	rXa[3] := X3;
	rXa[4] := X4;
	rXa[5] := X5;
	rXa[6] := X6;
	rXa[7] := X7;
	rXa[8] := X8;
	rXa[9] := X9;
	rXa[10] := X10;
	rXa[11] := X11;
	rXa[12] := X12;
	rXa[13] := X13;
	rXa[14] := X14;
	rXa[15] := X15;
	rXa[16] := X16;
	rXa[17] := X17;
	rXa[18] := X18;
	rXa[19] := X19;
	rXa[20] := X20;
	
	rYa[1] := Y1;
	rYa[2] := Y2;
	rYa[3] := Y3;
	rYa[4] := Y4;
	rYa[5] := Y5;
	rYa[6] := Y6;
	rYa[7] := Y7;	
	rYa[8] := Y8;
	rYa[9] := Y9;
	rYa[10] := Y10;
	rYa[11] := Y11;
	rYa[12] := Y12;
	rYa[13] := Y13;
	rYa[14] := Y14;
	rYa[15] := Y15;
	rYa[16] := Y16;
	rYa[17] := Y17;
	rYa[18] := Y18;
	rYa[19] := Y19;
	rYa[20] := Y20;

	//Calculate if value is out of boundaries	
	IF rTempUsed < rXa[1] THEN
		fScale20p := rYa[1];
	ELSIF rTempUsed > rXa[20] THEN
		fScale20p := rYa[20];
	ELSE	
		FOR iI := 1 TO 19 DO
			IF rTempUsed >= rXa[iI] AND rTempUsed <= rXa[iI + 1] THEN
				rM := (rYa[iI + 1] - rYa[iI])/(rXa[iI + 1]-rXa[iI]);
				fScale20p := rYa[iI] + rM * (rTempUsed - rXa[iI]);
				EXIT;
			END_IF
		END_FOR
	END_IF;

END_FUNCTION

// oaksLibrary/Beräkning/fScale2p
// Skalar om x till y med 2 punkter. Exempelvis för utekompensering.
FUNCTION fScale2p : REAL
VAR_INPUT
	 rX	 : ANY;	// Knyter man inget här används oaksGVL.rOutdoortemp som rX	
END_VAR
VAR_IN_OUT
	 Y1 : 	REAL;	
	 Y2:	REAL;	

	 X1:	REAL;	
	 X2:	REAL;	
END_VAR

VAR
 rTempUsed : REAL; // Uteluftstemperatur
 rXa : ARRAY[1..2] OF REAL;
 rYa : 	ARRAY[1..2] OF	REAL;
 rM :	REAL;	
 iI : 	INT;
END_VAR

	//Temp select
	rTempUsed := F_GetTempToUse(rX);

//Breakpoints must be ascending
	IF (X2 <= X1) THEN X2 := X1 + 0.1; END_IF
	//Copy data to array
	rXa[1] := X1;
	rXa[2] := X2;
	rYa[1] := Y1;
	rYa[2] := Y2;
	//Calculate if value is out of boundaries	
	IF rTempUsed < rXa[1] THEN
		fScale2p := rYa[1];
	ELSIF rTempUsed > rXa[2] THEN
		fScale2p := rYa[2];
	ELSE
		FOR iI := 1 TO 1 DO
			IF rTempUsed >= rXa[iI] AND rTempUsed <= rXa[iI + 1] THEN
				rM := (rYa[iI + 1] - rYa[iI])/(rXa[iI + 1]-rXa[iI]);
				fScale2p := rYa[iI] + rM * (rTempUsed - rXa[iI]);
				EXIT;
			END_IF
		END_FOR
	END_IF;

END_FUNCTION

// oaksLibrary/Beräkning/fScale2pInternalSetpoint
// Skalar om x till y med 2 punkter. Exempelvis för utekompensering.
FUNCTION fScale2pInternalSetpoint : REAL
VAR_INPUT
	 rX	 : ANY;	// Knyter man inget här används oaksGVL.rOutdoortemp som rX
	 Y1 : 	REAL;	
	 Y2:	REAL;	

	 X1:	REAL;	
	 X2:	REAL;	
END_VAR

VAR
 rTempUsed : REAL; // Uteluftstemperatur
 rXa : ARRAY[1..2] OF REAL;
 rYa : 	ARRAY[1..2] OF	REAL;
 rM :	REAL;	
 iI : 	INT;
END_VAR

	//Temp select
	rTempUsed := F_GetTempToUse(rX);

//Breakpoints must be ascending
	IF (X2 <= X1) THEN X2 := X1 + 0.1; END_IF
	//Copy data to array
	rXa[1] := X1;
	rXa[2] := X2;
	rYa[1] := Y1;
	rYa[2] := Y2;
	//Calculate if value is out of boundaries	
	IF rTempUsed < rXa[1] THEN
		fScale2pInternalSetpoint := rYa[1];
	ELSIF rTempUsed > rXa[2] THEN
		fScale2pInternalSetpoint := rYa[2];
	ELSE
		FOR iI := 1 TO 1 DO
			IF rTempUsed >= rXa[iI] AND rTempUsed <= rXa[iI + 1] THEN
				rM := (rYa[iI + 1] - rYa[iI])/(rXa[iI + 1]-rXa[iI]);
				fScale2pInternalSetpoint := rYa[iI] + rM * (rTempUsed - rXa[iI]);
				EXIT;
			END_IF
		END_FOR
	END_IF;

END_FUNCTION

// oaksLibrary/Beräkning/fScale3p
// Skalar om x till y med 2 punkter. Exempelvis för utekompensering.
FUNCTION fScale3p : REAL
VAR_INPUT
	 rX	 : ANY;	// Knyter man inget här används oaksGVL.rOutdoortemp som rX	
END_VAR
VAR_IN_OUT
	 Y1 : 	REAL;	
	 Y2:	REAL;	
	 Y3:	REAL;	

	 X1:	REAL;	
	 X2:	REAL;	
	 X3:	REAL;	
END_VAR

VAR
 rTempUsed : REAL; // Uteluftstemperatur
 rXa : ARRAY[1..3] OF REAL;
 rYa : 	ARRAY[1..3] OF	REAL;
 rM :	REAL;	
 iI : 	INT;
END_VAR

	//Temp select
	rTempUsed := F_GetTempToUse(rX);

//Breakpoints must be ascending
	IF (X2 <= X1) THEN X2 := X1 + 0.1; END_IF
	IF (X3 <= X2) THEN X3 := X2 + 0.1; END_IF
	//Copy data to array
	rXa[1] := X1;
	rXa[2] := X2;
	rXa[3] := X3;
	rYa[1] := Y1;
	rYa[2] := Y2;
	rYa[3] := Y3;
	//Calculate if value is out of boundaries	
	IF rTempUsed < rXa[1] THEN
		fScale3p := rYa[1];
	ELSIF rTempUsed > rXa[3] THEN
		fScale3p := rYa[3];
	ELSE
		FOR iI := 1 TO 2 DO
			IF rTempUsed >= rXa[iI] AND rTempUsed <= rXa[iI + 1] THEN
				rM := (rYa[iI + 1] - rYa[iI])/(rXa[iI + 1]-rXa[iI]);
				fScale3p := rYa[iI] + rM * (rTempUsed - rXa[iI]);
				EXIT;
			END_IF
		END_FOR
	END_IF;

END_FUNCTION

// oaksLibrary/Beräkning/fScale3pInternalSetpoint
// Skalar om x till y med 2 punkter. Exempelvis för utekompensering.
FUNCTION fScale3pInternalSetpoint : REAL
VAR_INPUT
	 rX	 : ANY;	// Knyter man inget här används oaksGVL.rOutdoortemp som rX
	 Y1 : 	REAL;	
	 Y2:	REAL;	
	 Y3:	REAL;

	 X1:	REAL;	
	 X2:	REAL;	
	 X3:	REAL;	
END_VAR

VAR
 rTempUsed : REAL; // Uteluftstemperatur
 rXa : ARRAY[1..3] OF REAL;
 rYa : 	ARRAY[1..3] OF	REAL;
 rM :	REAL;	
 iI : 	INT;
END_VAR

	//Temp select
	rTempUsed := F_GetTempToUse(rX);

//Breakpoints must be ascending
	IF (X2 <= X1) THEN X2 := X1 + 0.1; END_IF
	IF (X3 <= X2) THEN X3 := X2 + 0.1; END_IF
	//Copy data to array
	rXa[1] := X1;
	rXa[2] := X2;
	rXa[3] := X3;
	rYa[1] := Y1;
	rYa[2] := Y2;
	rYa[3] := Y3;
	//Calculate if value is out of boundaries	
	IF rTempUsed < rXa[1] THEN
		fScale3pInternalSetpoint := rYa[1];
	ELSIF rTempUsed > rXa[3] THEN
		fScale3pInternalSetpoint := rYa[3];
	ELSE
		FOR iI := 1 TO 2 DO
			IF rTempUsed >= rXa[iI] AND rTempUsed <= rXa[iI + 1] THEN
				rM := (rYa[iI + 1] - rYa[iI])/(rXa[iI + 1]-rXa[iI]);
				fScale3pInternalSetpoint := rYa[iI] + rM * (rTempUsed - rXa[iI]);
				EXIT;
			END_IF
		END_FOR
	END_IF;

END_FUNCTION

// oaksLibrary/Beräkning/fScale6p
// Skalar om x till y med 6 punkter. Exempelvis för utekompensering.
FUNCTION fScale6p : REAL
VAR_INPUT
	 rX	 : ANY;	// Knyter man inget här används oaksGVL.rOutdoortemp som rX	
END_VAR
VAR_IN_OUT
	 Y1 : 	REAL;	
	 Y2:	REAL;	
	 Y3:	REAL;	
	 Y4:	REAL;	
	 Y5:	REAL;	
	 Y6:	REAL;	
	 X1:	REAL;	
	 X2:	REAL;	
	 X3:	REAL;	
	 X4:	REAL;	
	 X5:	REAL;	
	 X6:	REAL;	
END_VAR
VAR
	rTempUsed : REAL; // Uteluftstemperatur
	 rXa : ARRAY[1..6] OF REAL;
	 rYa : 	ARRAY[1..6] OF	REAL;
	 rM :	REAL;	
	 iI : 	INT;
END_VAR

	//Temp select
	rTempUsed := F_GetTempToUse(rX);

//Breakpoints must be ascending
	IF (X2 <= X1) THEN X2 := X1 + 0.1; END_IF
	IF (X3 <= X2) THEN X3 := X2 + 0.1; END_IF
	IF (X4 <= X3) THEN X4 := X3 + 0.1; END_IF
	IF (X5 <= X4) THEN X5 := X4 + 0.1; END_IF
	IF (X6 <= X5) THEN X6 := X5 + 0.1; END_IF
 
	//Copy data to array
	rXa[1] := X1;
	rXa[2] := X2;
	rXa[3] := X3;
	rXa[4] := X4;
	rXa[5] := X5;
	rXa[6] := X6;
	rYa[1] := Y1;
	rYa[2] := Y2;
	rYa[3] := Y3;
	rYa[4] := Y4;
	rYa[5] := Y5;
	rYa[6] := Y6;

	//Calculate if value is out of boundaries	
	IF rTempUsed < rXa[1] THEN
		fScale6p := rYa[1];
	ELSIF rTempUsed > rXa[6] THEN
		fScale6p := rYa[6];
	ELSE	
		FOR iI := 1 TO 5 DO
			IF rTempUsed >= rXa[iI] AND rTempUsed <= rXa[iI + 1] THEN
				rM := (rYa[iI + 1] - rYa[iI])/(rXa[iI + 1]-rXa[iI]);
				fScale6p := rYa[iI] + rM * (rTempUsed - rXa[iI]);
				EXIT;
			END_IF
		END_FOR
	END_IF;

END_FUNCTION

// oaksLibrary/Beräkning/fScale6pInternalSetpoint
// Skalar om x till y med 6 punkter. Exempelvis för utekompensering. Ingen VAR-IN-OUT. 
FUNCTION fScale6pInternalSetpoint : REAL
VAR_INPUT
	 rX	 : ANY;	// Knyter man inget här används oaksGVL.rOutdoortemp som rX
	 y1 : 	REAL;	
	 y2:	REAL;	
	 y3:	REAL;	
	 y4:	REAL;	
	 y5:	REAL;	
	 y6:	REAL;	
	 x1:	REAL;	
	 x2:	REAL;	
	 x3:	REAL;	
	 x4:	REAL;	
	 x5:	REAL;	
	 x6:	REAL;	
END_VAR
VAR
	 rTempUsed : REAL; // Uteluftstemperatur
	 rXa : ARRAY[1..6] OF REAL;
	 rYa : 	ARRAY[1..6] OF	REAL;
	 rM :	REAL;	
	 iI : 	INT;
END_VAR

	//Temp select
	rTempUsed := F_GetTempToUse(rX);

//Breakpoints must be ascending
	IF (x2 <= x1) THEN x2 := x1 + 0.1; END_IF
	IF (x3 <= x2) THEN x3 := x2 + 0.1; END_IF
	IF (x4 <= x3) THEN x4 := x3 + 0.1; END_IF
	IF (x5 <= x4) THEN x5 := x4 + 0.1; END_IF
	IF (x6 <= x5) THEN x6 := x5 + 0.1; END_IF
 
	//Copy data to array
	rXa[1] := x1;
	rXa[2] := x2;
	rXa[3] := x3;
	rXa[4] := x4;
	rXa[5] := x5;
	rXa[6] := x6;
	rYa[1] := y1;
	rYa[2] := y2;
	rYa[3] := y3;
	rYa[4] := y4;
	rYa[5] := y5;
	rYa[6] := y6;

	//Calculate if value is out of boundaries	
	IF rTempUsed < rXa[1] THEN
		fScale6pInternalSetpoint := rYa[1];
	ELSIF rTempUsed > rXa[6] THEN
		fScale6pInternalSetpoint := rYa[6];
	ELSE	
		FOR iI := 1 TO 5 DO
			IF rTempUsed >= rXa[iI] AND rTempUsed <= rXa[iI + 1] THEN
				rM := (rYa[iI + 1] - rYa[iI])/(rXa[iI + 1]-rXa[iI]);
				fScale6pInternalSetpoint := rYa[iI] + rM * (rTempUsed - rXa[iI]);
				EXIT;
			END_IF
		END_FOR
	END_IF;

END_FUNCTION

// oaksLibrary/Beräkning/fScale7p
// Skalar om x till y med 6 punkter. Exempelvis för utekompensering.
FUNCTION fScale7p : REAL
VAR_INPUT
	 rX	 : ANY;	// Knyter man inget här används oaksGVL.rOutdoortemp som rX	
END_VAR
VAR_IN_OUT
	 Y1 : 	REAL;	
	 Y2:	REAL;	
	 Y3:	REAL;	
	 Y4:	REAL;	
	 Y5:	REAL;	
	 Y6:	REAL;	
	 Y7:	REAL;	
	 X1:	REAL;	
	 X2:	REAL;	
	 X3:	REAL;	
	 X4:	REAL;	
	 X5:	REAL;	
	 X6:	REAL;	
	 X7:	REAL;	
END_VAR
VAR
	rTempUsed : REAL; // Uteluftstemperatur
	 rXa : ARRAY[1..7] OF REAL;
	 rYa : 	ARRAY[1..7] OF	REAL;
	 rM :	REAL;	
	 iI : 	INT;
END_VAR

	//Temp select
	rTempUsed := F_GetTempToUse(rX);

//Breakpoints must be ascending
	IF (X2 <= X1) THEN X2 := X1 + 0.1; END_IF
	IF (X3 <= X2) THEN X3 := X2 + 0.1; END_IF
	IF (X4 <= X3) THEN X4 := X3 + 0.1; END_IF
	IF (X5 <= X4) THEN X5 := X4 + 0.1; END_IF
	IF (X6 <= X5) THEN X6 := X5 + 0.1; END_IF
	IF (X7 <= X6) THEN X7 := X6 + 0.1; END_IF
 
	//Copy data to array
	rXa[1] := X1;
	rXa[2] := X2;
	rXa[3] := X3;
	rXa[4] := X4;
	rXa[5] := X5;
	rXa[6] := X6;
	rXa[7] := X7;
	rYa[1] := Y1;
	rYa[2] := Y2;
	rYa[3] := Y3;
	rYa[4] := Y4;
	rYa[5] := Y5;
	rYa[6] := Y6;
	rYa[7] := Y7;

	//Calculate if value is out of boundaries	
	IF rTempUsed < rXa[1] THEN
		fScale7p := rYa[1];
	ELSIF rTempUsed > rXa[7] THEN
		fScale7p := rYa[7];
	ELSE	
		FOR iI := 1 TO 6 DO
			IF rTempUsed >= rXa[iI] AND rTempUsed <= rXa[iI + 1] THEN
				rM := (rYa[iI + 1] - rYa[iI])/(rXa[iI + 1]-rXa[iI]);
				fScale7p := rYa[iI] + rM * (rTempUsed - rXa[iI]);
				EXIT;
			END_IF
		END_FOR
	END_IF;

END_FUNCTION

// oaksLibrary/Beräkning/fScale7pInternalSetpoint
// Skalar om x till y med 6 punkter. Exempelvis för utekompensering. Ingen VAR-IN-OUT. 
FUNCTION fScale7pInternalSetpoint : REAL
VAR_INPUT
	 rX	 : ANY;	// Knyter man inget här används oaksGVL.rOutdoortemp som rX
	 y1 : 	REAL;	
	 y2:	REAL;	
	 y3:	REAL;	
	 y4:	REAL;	
	 y5:	REAL;	
	 y6:	REAL;	
	 y7:	REAL;	
	 x1:	REAL;	
	 x2:	REAL;	
	 x3:	REAL;	
	 x4:	REAL;	
	 x5:	REAL;	
	 x6:	REAL;	
	 x7:	REAL;	
END_VAR
VAR
	 rTempUsed : REAL; // Uteluftstemperatur
	 rXa : ARRAY[1..7] OF REAL;
	 rYa : 	ARRAY[1..7] OF	REAL;
	 rM :	REAL;	
	 iI : 	INT;
END_VAR

	//Temp select
	rTempUsed := F_GetTempToUse(rX);

//Breakpoints must be ascending
	IF (x2 <= x1) THEN x2 := x1 + 0.1; END_IF
	IF (x3 <= x2) THEN x3 := x2 + 0.1; END_IF
	IF (x4 <= x3) THEN x4 := x3 + 0.1; END_IF
	IF (x5 <= x4) THEN x5 := x4 + 0.1; END_IF
	IF (x6 <= x5) THEN x6 := x5 + 0.1; END_IF
	IF (x7 <= x6) THEN x7 := x6 + 0.1; END_IF
 
	//Copy data to array
	rXa[1] := x1;
	rXa[2] := x2;
	rXa[3] := x3;
	rXa[4] := x4;
	rXa[5] := x5;
	rXa[6] := x6;
	rXa[7] := x7;
	rYa[1] := y1;
	rYa[2] := y2;
	rYa[3] := y3;
	rYa[4] := y4;
	rYa[5] := y5;
	rYa[6] := y6;
	rYa[7] := y7;

	//Calculate if value is out of boundaries	
	IF rTempUsed < rXa[1] THEN
		fScale7pInternalSetpoint := rYa[1];
	ELSIF rTempUsed > rXa[7] THEN
		fScale7pInternalSetpoint := rYa[7];
	ELSE	
		FOR iI := 1 TO 6 DO
			IF rTempUsed >= rXa[iI] AND rTempUsed <= rXa[iI + 1] THEN
				rM := (rYa[iI + 1] - rYa[iI])/(rXa[iI + 1]-rXa[iI]);
				fScale7pInternalSetpoint := rYa[iI] + rM * (rTempUsed - rXa[iI]);
				EXIT;
			END_IF
		END_FOR
	END_IF;

END_FUNCTION

// oaksLibrary/Brand/fbFirealarm
FUNCTION_BLOCK fbFirealarm 
VAR_INPUT
	{attribute 'OPC.UA.DA' := '1'}
	V3 AT %I* : BOOL; //Larmingång~wp:[trendoptions]i:14400, t:1
	bInvert : BOOL;
	bAutoReset : BOOL := TRUE; // Auto-reset av larm
END_VAR
VAR_OUTPUT
	{attribute 'OPC.UA.DA' := '1'}
	AL AT %M*  : BOOL; //Utlöst centralt brandlarm~wp:[alarmoptions]p:1
END_VAR
VAR
	bInternalIndication : BOOL;
	fbAlarm1 : fbAlarm;
END_VAR

	IF NOT bInvert THEN
		bInternalIndication :=  V3;
	ELSE
		bInternalIndication := NOT V3;
	END_IF
		
	
	fbAlarm1(
	bInput:= bInternalIndication, 
	tAlarmDelay:= T#500MS, 
	bAutoReset:= bAutoReset, 
	bAlarmOutput=>AL );
	
	oaksgvl.bFireAlarm := AL;

END_FUNCTION_BLOCK

// oaksLibrary/Brand/fbFirealarmFailure
FUNCTION_BLOCK fbFirealarmFailure EXTENDS fbFirealarm
VAR_INPUT
	{attribute 'OPC.UA.DA' := '1'}
	V4 AT %I* : BOOL; //Larmingång fellarm~wp:[trendoptions]i:14400, t:1
	bInvertFailureAlarm : BOOL;
END_VAR
VAR_OUTPUT
	{attribute 'OPC.UA.DA' := '1'}
	AL1 AT %M*  : BOOL; //Fellarm brandlarmscentral~wp:[alarmoptions]p:2
END_VAR
VAR
	bInternalIndicationFailureAlarm : BOOL;
	fbAlarm2 : fbAlarm;
END_VAR

	SUPER^();

	IF NOT bInvert THEN
		bInternalIndicationFailureAlarm :=  V4;
	ELSE
		bInternalIndicationFailureAlarm := NOT V4;
	END_IF
		
	fbAlarm1(
	bInput:= bInternalIndicationFailureAlarm, 
	tAlarmDelay:= T#500MS, 
	bAutoReset:= bAutoReset, 
	bAlarmOutput=>AL1 );

END_FUNCTION_BLOCK

// oaksLibrary/Brand/fbFireDamper
//Oaks AB 2020-06-10
//Funktionsblock för styrning av brandspjäll med öppet/stängt indikering (stänger på fjäder). 
FUNCTION_BLOCK fbFireDamper
VAR_INPUT
bMotion : BOOL; //Motionskörning
bSafe : BOOL; //Säkerhetsvillkor
tAlarmDelay : TIME := T#180S; // Larmfördröjning
END_VAR
VAR_OUTPUT
{attribute 'OPC.UA.DA' := '1'}
CMD AT %Q* : BOOL; //Manöver~wp:[trendoptions]i:14400, t:1
{attribute 'OPC.UA.DA' := '1'}
V0 AT %I* : BOOL; //Stängtindikering~wp:[trendoptions]i:14400, t:1
{attribute 'OPC.UA.DA' := '1'}
V1 AT %I* : BOOL; //Öppetindikering~wp:[trendoptions]i:14400, t:1
{attribute 'OPC.UA.DA' := '1'}
AL AT %M* : BOOL; //Spjällfel~wp:
{attribute 'OPC.UA.DA' := '1'}
PV4 AT %M* : BOOL; //Motionskörning aktiv~wp:[trendoptions]i:14400, t:1
END_VAR
VAR
	itemp : int;
	SR_1: SR;
	fbStartPulse: TP; // Startpuls	
	fbMotionTime: TP; // Håller en puls under motionskörning
	fbStopMotion: F_TRIG;
	fbAlarm1: fbAlarm;
	bAlarm: BOOL;
	IN: INT;
END_VAR

//Aktivera motionering på positiv flank (SET)
fbStartPulse(IN:= bMotion, PT:= T#1S, Q=> , ET=> ); //Startar en puls
//Hållkrets
SR_1(
SET1:= fbStartPulse.Q, 
RESET:= fbStopMotion.Q OR V0, 
Q1=> PV4
);

//Avaktivera motionering (RESET)
fbMotionTime(IN:= fbStartPulse.Q, PT:= T#300S, Q=> , ET=> ); //Startar en puls
fbStopMotion(CLK:= fbMotionTime.Q, Q=> ); // Reset då pulstid gått ut

//Utgång
CMD := bSafe AND NOT PV4;

//Larm
bAlarm := (NOT CMD AND NOT V0) OR (CMD AND NOT V1);

fbAlarm1(bInput:=bAlarm , tAlarmDelay:=tAlarmDelay , bAutoReset:= TRUE, bAlarmOutput=> AL);

END_FUNCTION_BLOCK

// oaksLibrary/Brand/fbFireDamperEvac
//Oaks AB 2020-06-10
//Funktionsblock för styrning av rökevakueringsspjäll med öppet/stängt indikering (öppnar på fjäder). 
FUNCTION_BLOCK fbFireDamperEvac
VAR_INPUT
bMotion : BOOL; //Motionskörning
bSafe : BOOL; //Säkerhetsvillkor
tAlarmDelay : TIME := T#180S; // Larmfördröjning
END_VAR
VAR_OUTPUT
	{attribute 'OPC.UA.DA' := '1'}
	CMD AT %Q* : BOOL; //Manöver~wp:[trendoptions]i:14400, t:1
	{attribute 'OPC.UA.DA' := '1'}
	V1 AT %I* : BOOL; //Öppetindikering~wp:[trendoptions]i:14400, t:1
	{attribute 'OPC.UA.DA' := '1'}
	V0 AT %I* : BOOL; //Stängtindikering~wp:[trendoptions]i:14400, t:1
	{attribute 'OPC.UA.DA' := '1'}
	AL AT %M* : BOOL; //Spjällfel~wp:
	{attribute 'OPC.UA.DA' := '1'}
	PV4 AT %M* : BOOL; //Motionskörning aktiv~wp:[trendoptions]i:14400, t:1
END_VAR
VAR
	itemp : int;
	SR_1: SR;
	fbStartPulse: TP; //Startpuls	
	fbMotionTime: TP; //Håller en puls under motionskörning
	fbStopMotion: F_TRIG;
	fbAlarm1: fbAlarm;
	bAlarm: BOOL;
	IN: INT;
END_VAR

//Aktivera motionering på positiv flank (SET)
fbStartPulse(IN:= bMotion, PT:= T#1S, Q=> , ET=> ); //Startar en puls

//Hållkrets
SR_1(
SET1:= fbStartPulse.Q, 
RESET:= fbStopMotion.Q OR V1, 
Q1=> PV4
);

//Avaktivera motionering (RESET)
fbMotionTime(IN:= fbStartPulse.Q, PT:= T#300S, Q=> , ET=> ); //Startar en puls
fbStopMotion(CLK:= fbMotionTime.Q, Q=> ); // Reset då pulstid gått ut

//Utgång
CMD := bSafe AND NOT PV4;

//Larm
bAlarm := (NOT CMD AND NOT V1) OR (CMD AND NOT V0);

fbAlarm1(bInput:=bAlarm , tAlarmDelay:=tAlarmDelay , bAutoReset:= TRUE, bAlarmOutput=> AL);

END_FUNCTION_BLOCK

// oaksLibrary/Brand/fbFiredamperExercise
// Block för global pumpmotion. V i blocket sätter internt i blocket den globala variabeln oaksGVL.bPumpMotion. 
// oaksGVL.bPumpMotion finns knuten i fbMotor och aktiverar pumpmotion om bPumpmotionConfig i respektive fbMotor-instans är till.
FUNCTION_BLOCK fbFiredamperExercise
VAR_INPUT
	{attribute 'OPC.UA.DA' := '1'}
	M AT %M*  : BOOL; //Test brandspjäll~wp:[trendoptions]i:14400, t:1
END_VAR
VAR_OUTPUT
	{attribute 'OPC.UA.DA' := '1'}
	V AT %M*  : BOOL; //Brandspjällsmotionering aktiv~wp:[trendoption]i:300[trendoptions]i:14400, t:1
	{attribute 'OPC.UA.DA' := '1'}
	PV AT %M*  : STRING; //Dag för motionering~wp:
	{attribute 'OPC.UA.DA' := '1'}
	PV1 AT %M* : INT; //Tid för motionering~wp:[format]00:00
END_VAR
VAR
	stTime		: tc2_ba.TIMESTRUCT;
	nActualDayCase	: INT;
	nActualHour 	: INT;
	nActualMinute 	: INT;
	
	FB_BA_GetTime01 : tc2_ba.FB_BA_GetTime; 
	FB_BA_ExtTiSt01 : tc2_ba.FB_BA_ExtTiSt;	
	
	itemp : int;
	nTime : INT; // Internvariabel aktuell tid (nActualHour+nActualMinute)
	
	bDay : BOOL; // Internvariabel blir TRUE om inställd dag är lika med aktuell dag
	bTime : BOOL; // Internvariabel blir TRUE om inställd tid är lika med aktuell tid
	fbHandsetToN: TON;
END_VAR
VAR_INPUT PERSISTENT
	{attribute 'OPC.UA.DA' := '1'}
	SP1 AT %M*  : INT:=1; //Dag för brandspjällsmotionering (0 = Söndag 1 = Måndag 2 = Tisdag..6 = Söndag~wp:
	{attribute 'OPC.UA.DA' := '1'}
	SP2 AT %M*  : INT:=1000; //Tid för brandspjällsmotionering~wp:[format]00:00[engmin]0[engmax]2400
END_VAR

	IF SP1 < 0 OR  SP1>6 THEN
		SP1 := 1;
	END_IF
	
	IF SP2 < 0 OR  SP2>2359 THEN
		SP2 := 1200;
	END_IF
	
	

	FB_BA_GetTime01(bEn :=TRUE);	
	stTime := FB_BA_GetTime01.stSysTi;

	nActualDayCase :=WORD_TO_INT (stTime.wDayOfWeek);
	nActualHour :=WORD_TO_INT (stTime.wHour)*100;
	nActualMinute :=WORD_TO_INT (stTime.wMinute);
	
	// nActualHour+nActualMinute
	
	nTime := nActualHour+nActualMinute;
	
	bDay := nActualDayCase = SP1;
	bTime := nTime = SP2;
	
	fbHandsetToN.PT := T#1M;
	fbHandsetToN(IN:=M);
	
	IF fbHandsetToN.Q THEN 
		M := FALSE;
	END_IF
	
	
	V := (bDay AND bTime) OR M;

	//För visning i Webport	
	PV1:= SP2;

	CASE SP1 OF
		0: PV:= 'Söndag';
		1: PV:= 'Måndag';
		2: PV:= 'Tisdag';
		3: PV:= 'Onsdag';
		4: PV:= 'Torsdag';
		5: PV:= 'Fredag';
		6: PV:= 'Lördag';
	END_CASE

END_FUNCTION_BLOCK

// oaksLibrary/Utsignal DO_AO/Motorer/fbMotor
// "Motorblock" för digital utsignal med driftsvar/summalarm med möjlighet att handställa utsignal. Larmar vid handställning eller utebliven driftindikering/summalarm.
FUNCTION_BLOCK fbMotor
VAR_INPUT
	bStart : BOOL; // Startvillkor
	bPumpmotionConfig : BOOL; // TRUE = global funktion för pumpmotion används. Kräver att bSafe är till för att pumpmotion ska kunna köras. Kräver att ett block av typen fbPumpmotion deklareras och körs.
	bServiceStop : BOOL; // Serviceomkopplare utgång går från om denna ingång är till
	bSafe: BOOL; // Säkerhetsvillkor - Blockerar utsignal i autoläge samt blockerar handställning. Måste vara TRUE för att block ska kunna köras. 
	bSumAlarmConfig : BOOL; // TRUE = summalarm FALSE = driftindikering
	bInputInvert :BOOL; // invertering av digtal insignal
	bAutoReset : BOOL := TRUE; // auto-reset utav driftfel
	bHandsetBlock : BOOL; // Används för blockering av handställning utan att blockera utsignal i autoläge. OBS! - För säkerhetsvillkor se ingång bSafe!
	tAlarmDelay : TIME := T#3S; // Larmfördröjning
	tStartDelay : TIME := T#0S; // Startfördröjning
	tStopDelay : TIME := T#0S; // Stoppfördröjning
	bExternalIndication : BOOL := TRUE; // Här knyts eventuell tryckvakt eller liknande för att exempelvis få driftfel vid bortfall av tryck
	bExternalIndicationOnly : BOOL := FALSE; //Används istället för IO-knytning för tex driftindikering från Metz
	{attribute 'OPC.UA.DA' := '1'}
	RST AT %M* : BOOL := FALSE; //Nollställ drifttid~wp: 
END_VAR
VAR_OUTPUT
	{attribute 'OPC.UA.DA' := '1'}
	CMD AT %Q*  : BOOL; //Utsignal~wp:[trendoptions]i:14400, t:1
	{attribute 'OPC.UA.DA' := '1'}
	V AT %M*   : BOOL; //Driftindikering~wp:[trendoptions]i:14400, t:1
	{attribute 'OPC.UA.DA' := '1'}
	AL AT %M* : BOOL; //Driftfel~wp:
	{attribute 'OPC.UA.DA' := '1'}
	AL8 AT %M* : BOOL; //Utsignal handställd~wp:[alarmoptions]p:3
	bAlarmOutput : BOOL; // internvariabel larm , används för knytning till exempelvis aggregatsblock
	bHandsetOutput : BOOL; // internvariabel handställning, används för knytning till exempelvis aggregatsblock
	{attribute 'OPC.UA.DA' := '1'}
	PV8 AT %M* : STRING; //Konfiguration digital ingång~wp:
	{attribute 'OPC.UA.DA' := '1'}
	PV7 AT %M* : UDINT; //Drifttid~wp:[unit]timmar[format]0[trendoptions]i:300
	STATE1 AT %M* : STRING; //Status IO-modul~wp:
	tStartDelayRemaining : TIME; // Aktuell  återstående tid startfördröjning
	tStopDelayRemaining : TIME; // Aktuell återstående tid stoppfördröjning
	bStopDelay : BOOL; //Stopp fördröjning aktiverad (för tex. stopp kylmaskin)
END_VAR
VAR
	bInternalStart : BOOL;
	bIndication AT %I* : BOOL; // om bSumAlarmConfig = TRUE summalarmsingång annars driftindikering.
	bProcessedIndication :BOOL; 
	bAlarm : BOOL;
	fbAlarm1 : fbAlarm;
	bPumpMotionStart : BOOL; // starta pumpmotion
	
	fbAlarm2 : fbAlarm; // Larm handställning
	fbStartDelay: TON; // Startfördröjning
	fbStopDelay: TOF; // Stoppfördröjning
	fbOperatingHours_1: fbOperatingHours;
	
	//Handställningsvariabler från IO
	TI_bStateAuto AT %I* :BOOL :=TRUE; //Status Auto/Manuell
	TI_bStateRelay AT %I* :BOOL :=FALSE; //Status reläutgång
	bIOManual : BOOL;
	
END_VAR
VAR_INPUT PERSISTENT
	{attribute 'OPC.UA.DA' := '1'}
	M AT %M* : BOOL; //Handställning~wp:[trendoptions]i:14400, t:1
	{attribute 'OPC.UA.DA' := '1'}
	MCMD AT %M* : BOOL; //Styrsignal handställning~wp:[trendoptions]i:14400, t:1
END_VAR

	fbAlarm2(bInput:=M OR NOT TI_bStateAuto, tAlarmDelay:= , bAutoReset:=TRUE , bAlarmOutput=>AL8 );
	
	//Välj om IO eller bExternalIndication skall användas för indikering
	IF NOT bExternalIndicationOnly THEN
		IF bInputInvert THEN
			bProcessedIndication := NOT bIndication AND bExternalIndication;
		ELSE
			bProcessedIndication := bIndication AND bExternalIndication;
		END_IF
	ELSE
		IF bInputInvert THEN
			bProcessedIndication := NOT bExternalIndication;
		ELSE
			bProcessedIndication := bExternalIndication;
		END_IF
	END_IF
		
	IF bSumAlarmConfig THEN
		V := bProcessedIndication AND CMD;
	ELSE
		V := bProcessedIndication;
	END_IF

	//Handställning
	IF NOT bSafe OR bHandsetBlock OR bServiceStop THEN
		M := FALSE;
	END_IF;
			
	IF bSumAlarmConfig AND bInputInvert THEN
		PV8 := 'Summalarm NO';
	ELSIF bSumAlarmConfig AND NOT bInputInvert THEN 
		PV8 := 'Summalarm NC'; 
	ELSIF NOT bSumAlarmConfig AND bInputInvert THEN
		PV8 := 'Driftindikering inverterad';
	ELSE
		PV8 := 'Driftindikering';
	END_IF
		
	//Start-/stoppfördröjning
    fbStartDelay(IN:=bStart , PT:=tStartDelay , Q=> , ET=> );
	fbStopDelay(IN:=fbStartDelay.Q, PT:=tStopDelay , Q=> , ET=> );
	
	tStopDelayRemaining := mTimeRemainingTof(fbStopDelay);
	tStartDelayRemaining := mTimeRemainingTon(fbStartDelay);
	
	bInternalStart := fbStopDelay.Q;
	
	IF tStopDelayRemaining < tStopDelay AND tStopDelayRemaining <> t#0s THEN
		bStopDelay := TRUE;
	ELSE
		bStopDelay := FALSE;
	END_IF
		
	// Startar pump om motor är konfigurerad för global pumpmotion 
	IF bPumpmotionConfig THEN
		bPumpMotionStart := oaksGVL.bPumpMotion;
	ELSE
		bPumpMotionStart := FALSE;
	END_IF
	
	//Manuell omkopplare IO-modul
	bIOManual := fKx2652State(bAuto := TI_bStateAuto, bRelayStatus := TI_bStateRelay, sState => STATE1);
	
	IF NOT TI_bStateAuto THEN
		CMD := bIOManual;
	ELSE
		CMD := ((((bInternalStart OR bPumpMotionStart) AND NOT M) OR (M AND MCMD)) AND bSafe AND NOT bServiceStop) OR bIOManual;	
	END_IF
	
	IF bSumAlarmConfig THEN
		bAlarm := NOT bProcessedIndication;
	ELSE
		bAlarm := V XOR CMD;
	END_IF

	
	fbAlarm1(bInput:=bAlarm , tAlarmDelay:=tAlarmDelay , bAutoReset:=bAutoReset , bAlarmOutput=> AL);
	
	bAlarmOutput := AL;
	bHandsetOutput := M;
	
	//Drifttidsmätning
	fbOperatingHours_1(bEnable:= V, bReset:= RST, rOperatingHours=> PV7 );

METHOD PUBLIC mStartDelayRemaining : STRING
VAR_INPUT
	sStatusString : STRING;
END_VAR
VAR
	tTime : TIME; 
END_VAR
	tTime := mTimeRemainingTon(fbStartDelay);
	
	
	IF tTime > T#0S AND tTime < fbStartDelay.PT AND NOT bPumpMotionStart AND NOT M AND TI_bStateAuto  THEN
 		mStartDelayRemaining := CONCAT(sStatusString,CONCAT(INT_TO_STRING(TIME_TO_INT(tTime/1000)), ' s'));
	ELSE
		mStartDelayRemaining := ' ';
	END_IF
END_METHOD

METHOD PUBLIC mStopDelayRemaining : STRING
VAR_INPUT
	sStatusString : STRING;
END_VAR
VAR
	tTime : TIME; 
END_VAR
	tTime := mTimeRemainingTof(fbStopDelay);
	
	
	IF tTime > T#0S AND tTime < fbStopDelay.PT AND NOT bPumpMotionStart AND NOT M AND TI_bStateAuto  THEN
 		mStopDelayRemaining := CONCAT(sStatusString,CONCAT(INT_TO_STRING(TIME_TO_INT(tTime/1000)), ' s'));
	ELSE
		mStopDelayRemaining := ' ';
	END_IF
END_METHOD

METHOD PROTECTED mTimeRemainingTof : TIME
VAR_IN_OUT
	fbTof : TOF;
END_VAR
mTimeRemainingTof := fbTof.PT - fbTof.ET;
END_METHOD

METHOD PROTECTED mTimeRemainingTon : TIME
VAR_IN_OUT
	fbTon : TON;
END_VAR
mTimeRemainingTon := fbTon.PT - fbTon.ET;
END_METHOD

END_FUNCTION_BLOCK

// oaksLibrary/Utsignal DO_AO/fKx2652State
FUNCTION fKx2652State : BOOL
VAR_INPUT
	bAuto : BOOL; //IO-modul i läge AUTO
	bRelayStatus : BOOL; //IO-modul relästatus
END_VAR
VAR
END_VAR

VAR_OUTPUT
	sState : STRING;
END_VAR

IF NOT bAUTO AND bRelayStatus = TRUE THEN
	fKx2652State := TRUE;
	sState := 'Handställd till ON på IO-enhet';
ELSIF  NOT bAUTO AND bRelayStatus = FALSE THEN
	fKx2652State := FALSE;
	sState := 'Handställd till OFF på IO-enhet';
ELSE
	fKx2652State := FALSE;
	sState := ' ';
END_IF

END_FUNCTION

